ABB RAPID module: ST1606_R04_SWP_2.mod

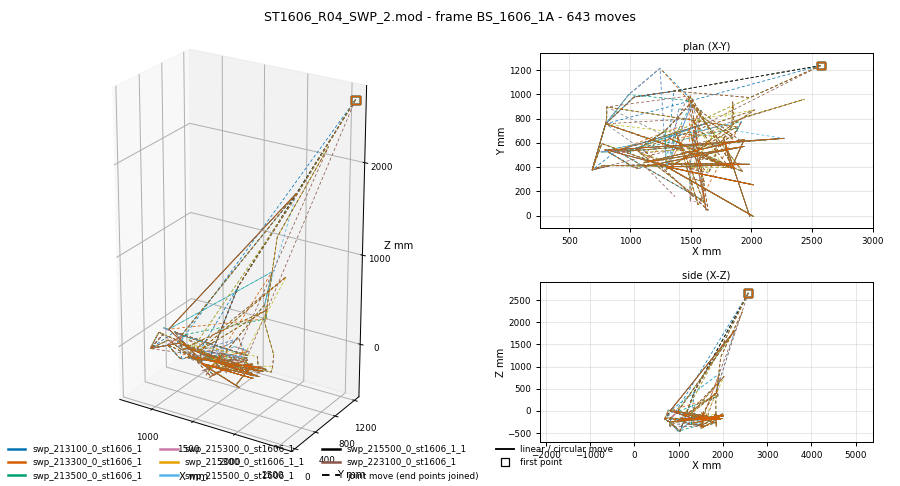
[picture p0: tool path of ST1606_R04_SWP_2.mod in frame BS_1606_1A, 643 of 1025 moves have a stored position in this frame; points joined in program order, loops and branches not executed]
MODULE ST1606_R04_SWP_2
CONST robtarget LHP_285:=[[1303.72,403.68,-203.75],[0.635635,0.00179403,0.00318194,-0.771981],[-1,-1,-1,0],[9E+09,9E+09,9E+09,9E+09,9E+09,9E+09]];
CONST robtarget LHP_275:=[[1301.19,402.05,-200.09],[0.6354,0.000830935,0.00305671,-0.772177],[-1,-1,-1,0],[9E+09,9E+09,9E+09,9E+09,9E+09,9E+09]];
CONST robtarget LHP_295:=[[1301.18,402.05,-200.09],[0.635399,0.000829977,0.00305677,-0.772177],[-1,-1,-1,0],[9E+09,9E+09,9E+09,9E+09,9E+09,9E+09]];
CONST robtarget LHP_270:=[[767.48,594.20,-155.47],[0.511232,-0.0380294,0.0384775,-0.857738],[-1,-1,-1,0],[9E+09,9E+09,9E+09,9E+09,9E+09,9E+09]];
CONST robtarget LHP_35:=[[946.51,280.68,-61.37],[0.681512,-0.0530703,0.0236717,-0.729496],[-1,-1,-1,0],[9E+09,9E+09,9E+09,9E+09,9E+09,9E+09]];
CONST robtarget LHP_76:=[[1001.84,541.68,-25.00],[0.296784,-0.0658707,0.043797,-0.951663],[-1,-1,0,0],[9E+09,9E+09,9E+09,9E+09,9E+09,9E+09]];
CONST robtarget LHP_80:=[[888.28,533.44,-4.12],[0.256081,-0.0828864,0.058088,-0.961342],[-1,-1,0,0],[9E+09,9E+09,9E+09,9E+09,9E+09,9E+09]];
CONST robtarget LHP_90:=[[990.54,532.98,-17.68],[0.294359,-0.0710943,0.0347938,-0.952411],[-1,-1,0,0],[9E+09,9E+09,9E+09,9E+09,9E+09,9E+09]];
CONST robtarget LHP_86:=[[888.43,535.56,-4.02],[0.256121,-0.0829008,0.0580729,-0.961331],[-1,-1,0,0],[9E+09,9E+09,9E+09,9E+09,9E+09,9E+09]];
CONST robtarget LHP_96:=[[1001.89,531.58,-24.98],[0.296786,-0.0658745,0.0437906,-0.951662],[-1,-1,0,0],[9E+09,9E+09,9E+09,9E+09,9E+09,9E+09]];
CONST robtarget LHP_120:=[[888.43,534.97,-4.06],[0.256117,-0.0828895,0.0580877,-0.961332],[-1,-1,0,0],[9E+09,9E+09,9E+09,9E+09,9E+09,9E+09]];
CONST robtarget LHP_130:=[[976.30,531.44,-18.23],[0.289518,-0.0722185,0.03693,-0.95373],[-1,-1,0,0],[9E+09,9E+09,9E+09,9E+09,9E+09,9E+09]];
CONST robtarget LHP_106:=[[818.07,526.79,7.37],[0.226549,-0.0825481,0.052721,-0.969062],[-1,-1,0,0],[9E+09,9E+09,9E+09,9E+09,9E+09,9E+09]];
CONST robtarget LHP_140:=[[813.23,540.09,5.50],[0.203616,-0.0600557,0.0553882,-0.975636],[-1,-1,0,0],[9E+09,9E+09,9E+09,9E+09,9E+09,9E+09]];
CONST robtarget LHP_305:=[[1315.92,428.20,-139.09],[0.644633,0.00162574,0.00306103,-0.764485],[-1,-1,-1,0],[9E+09,9E+09,9E+09,9E+09,9E+09,9E+09]];
CONST robtarget LHP_95:=[[1137.13,401.53,-148.24],[0.465302,0.0650512,0.0937079,-0.877771],[-1,-1,-1,0],[9E+09,9E+09,9E+09,9E+09,9E+09,9E+09]];
CONST robtarget LHP_30:=[[810.70,415.20,9.23],[0.639806,-0.0807189,0.0295354,-0.763715],[-1,-1,-1,0],[9E+09,9E+09,9E+09,9E+09,9E+09,9E+09]];
CONST robtarget LHP_75:=[[1074.27,512.60,-33.94],[0.333599,-0.0675086,0.0283306,-0.939868],[-1,-1,0,0],[9E+09,9E+09,9E+09,9E+09,9E+09,9E+09]];
CONST robtarget LHP_60:=[[1486.65,949.59,-335.01],[0.314,0.0992422,0.101035,-0.938801],[-1,-1,0,0],[9E+09,9E+09,9E+09,9E+09,9E+09,9E+09]];
CONST robtarget LHP_62:=[[1903.50,403.96,-168.40],[0.688588,0.0102129,0.00768242,-0.72504],[-1,-1,-1,0],[9E+09,9E+09,9E+09,9E+09,9E+09,9E+09]];
CONST robtarget LHP_061:=[[1899.73,616.36,-175.94],[0.688576,0.010205,0.00768425,-0.725052],[-1,-1,-1,0],[9E+09,9E+09,9E+09,9E+09,9E+09,9E+09]];
CONST robtarget LHP_602:=[[1726.06,605.49,-175.95],[0.68856,0.0102045,0.00768354,-0.725067],[-1,-1,-1,0],[9E+09,9E+09,9E+09,9E+09,9E+09,9E+09]];
CONST robtarget LHP_079:=[[2016.26,-5.68,-78.35],[0.747483,0.000532313,0.000430293,-0.664281],[-1,-1,-1,0],[9E+09,9E+09,9E+09,9E+09,9E+09,9E+09]];
CONST robtarget LHP_0792:=[[1914.27,375.53,-160.96],[0.711937,0.00638954,0.00588801,-0.702189],[-1,-1,-1,0],[9E+09,9E+09,9E+09,9E+09,9E+09,9E+09]];
CONST robtarget LHP_65:=[[1317.44,742.66,-303.72],[0.355107,0.0744104,0.10019,-0.926458],[-1,-1,0,0],[9E+09,9E+09,9E+09,9E+09,9E+09,9E+09]];
CONST robtarget LHP_85:=[[1629.29,310.10,-175.34],[0.669574,0.0105491,-0.00428905,-0.742658],[-1,0,-1,0],[9E+09,9E+09,9E+09,9E+09,9E+09,9E+09]];
CONST robtarget LHP_315:=[[1770.47,642.52,-185.25],[0.687362,-0.000165211,-0.0154473,-0.726151],[-1,0,-1,0],[9E+09,9E+09,9E+09,9E+09,9E+09,9E+09]];
CONST robtarget LHP_325:=[[1942.15,629.05,-193.52],[0.692101,-6.80423E-05,-0.0154578,-0.721635],[-1,0,-1,0],[9E+09,9E+09,9E+09,9E+09,9E+09,9E+09]];
CONST robtarget LHP_335:=[[1942.18,570.86,-193.52],[0.673118,-0.00046509,-0.0154488,-0.739373],[-1,0,-1,0],[9E+09,9E+09,9E+09,9E+09,9E+09,9E+09]];
CONST robtarget LHP_345:=[[1903.37,431.47,-166.61],[0.699368,0.00456834,-0.0108725,-0.714664],[-1,0,-1,0],[9E+09,9E+09,9E+09,9E+09,9E+09,9E+09]];
CONST robtarget LHP_355:=[[1863.39,397.38,-157.88],[0.649959,0.00383079,-0.0111584,-0.759877],[-1,0,-1,0],[9E+09,9E+09,9E+09,9E+09,9E+09,9E+09]];
CONST robtarget LHP_365:=[[1863.47,385.43,-144.48],[0.649789,-0.0155667,-0.0338777,-0.7592],[-1,0,-1,0],[9E+09,9E+09,9E+09,9E+09,9E+09,9E+09]];
CONST robtarget LHP_280:=[[2016.33,-5.64,-99.38],[0.747492,0.000549922,0.000436579,-0.664271],[-1,-1,-1,0],[9E+09,9E+09,9E+09,9E+09,9E+09,9E+09]];
CONST robtarget LHP_290:=[[2016.31,254.27,-112.69],[0.752523,0.000550496,0.000440421,-0.658565],[-1,-1,-1,0],[9E+09,9E+09,9E+09,9E+09,9E+09,9E+09]];
CONST robtarget LHP_300:=[[1984.86,424.01,-175.49],[0.757242,0.000550801,0.000441944,-0.653134],[-1,-1,-1,0],[9E+09,9E+09,9E+09,9E+09,9E+09,9E+09]];
CONST robtarget LHP_375:=[[1628.09,45.58,-117.32],[0.667896,0.00169065,-0.00043216,-0.744252],[-1,0,-1,0],[9E+09,9E+09,9E+09,9E+09,9E+09,9E+09]];
CONST robtarget LHP_385:=[[1611.54,278.38,-117.33],[0.667901,0.00169334,-0.000433516,-0.744248],[-1,0,-1,0],[9E+09,9E+09,9E+09,9E+09,9E+09,9E+09]];
CONST robtarget LHP_116:=[[1000.78,413.85,-25.10],[0.394135,-0.0875222,0.0272439,-0.91447],[-1,-1,0,0],[9E+09,9E+09,9E+09,9E+09,9E+09,9E+09]];
CONST robtarget LHP_150:=[[1561.93,87.92,-128.43],[0.625297,0.0429298,0.0210226,-0.778921],[-1,-1,-1,0],[9E+09,9E+09,9E+09,9E+09,9E+09,9E+09]];
CONST robtarget LHP_395:=[[1629.22,373.82,-175.87],[0.62292,0.0114274,-0.00461499,-0.782189],[-1,0,-1,0],[9E+09,9E+09,9E+09,9E+09,9E+09,9E+09]];
CONST robtarget LHP_405:=[[1666.92,623.72,-173.59],[0.685638,0.0117691,-0.00364924,-0.727838],[-1,0,-1,0],[9E+09,9E+09,9E+09,9E+09,9E+09,9E+09]];
CONST robtarget LHP_415:=[[1910.33,618.10,-173.56],[0.724769,0.0119478,-0.00298906,-0.688882],[-1,0,-1,0],[9E+09,9E+09,9E+09,9E+09,9E+09,9E+09]];
CONST robtarget LHP_425:=[[1929.29,361.85,-152.34],[0.724775,0.0119437,-0.00298739,-0.688875],[-1,0,-1,0],[9E+09,9E+09,9E+09,9E+09,9E+09,9E+09]];
CONST robtarget LHP_435:=[[1816.72,397.75,-147.92],[0.816486,0.00152322,-0.000785194,-0.577362],[-1,0,-1,0],[9E+09,9E+09,9E+09,9E+09,9E+09,9E+09]];
CONST robtarget LHP_310:=[[1987.44,-5.82,-69.73],[0.747483,0.000551369,0.000433351,-0.664281],[-1,-1,-1,0],[9E+09,9E+09,9E+09,9E+09,9E+09,9E+09]];
CONST robtarget LHP_445:=[[1643.36,44.45,-93.66],[0.669275,0.0117171,-0.00391081,-0.742912],[-1,0,-1,0],[9E+09,9E+09,9E+09,9E+09,9E+09,9E+09]];
CONST robtarget LHP_081:=[[1770.69,382.20,-42.12],[0.747485,0.000553614,0.00043516,-0.664279],[-1,-1,-1,0],[9E+09,9E+09,9E+09,9E+09,9E+09,9E+09]];
CONST robtarget LHP_320:=[[1834.77,390.06,-64.76],[0.679356,0.0474033,0.0375445,-0.731313],[-1,-1,-1,0],[9E+09,9E+09,9E+09,9E+09,9E+09,9E+09]];
CONST robtarget LHP_088:=[[1834.77,390.06,-64.76],[0.679356,0.0474033,0.0375445,-0.731313],[-1,-1,-1,0],[9E+09,9E+09,9E+09,9E+09,9E+09,9E+09]];
CONST robtarget LHP_97:=[[1624.62,82.13,-48.66],[0.622006,0.00520638,0.00406435,-0.782985],[-1,-1,-1,0],[9E+09,9E+09,9E+09,9E+09,9E+09,9E+09]];
LOCAL CONST robtarget LHP_089:=[[1624.62,82.13,-48.66],[0.622006,0.00520701,0.00406451,-0.782985],[-1,-1,-1,0],[9E+09,9E+09,9E+09,9E+09,9E+09,9E+09]];
CONST robtarget LHP_99:=[[1624.61,82.13,-48.66],[0.622006,0.00520638,0.00406435,-0.782985],[-1,-1,-1,0],[9E+09,9E+09,9E+09,9E+09,9E+09,9E+09]];
CONST robtarget LHP_109:=[[1624.62,82.13,-48.66],[0.622006,0.00520677,0.00406445,-0.782985],[-1,-1,-1,0],[9E+09,9E+09,9E+09,9E+09,9E+09,9E+09]];
CONST robtarget G0216022538BPS0:=[[2172.49,515.89,-41.57],[0.756815,0.0088806,0.00204198,-0.653566],[-1,-1,-1,0],[9E+09,9E+09,9E+09,9E+09,9E+09,9E+09]];
CONST robtarget LHP_40:=[[809.47,413.89,9.27],[0.637646,-0.0807527,0.029297,-0.765525],[-1,-1,-1,0],[9E+09,9E+09,9E+09,9E+09,9E+09,9E+09]];
CONST robtarget LHP_160:=[[1610.65,106.32,-46.18],[0.687963,0.00231302,0.000740632,-0.725741],[-1,-1,-1,0],[9E+09,9E+09,9E+09,9E+09,9E+09,9E+09]];
CONST robtarget LHP_126:=[[1076.78,394.51,-236.89],[0.363169,0.0511528,0.105229,-0.924347],[-1,-1,0,0],[9E+09,9E+09,9E+09,9E+09,9E+09,9E+09]];
CONST robtarget LHP_170:=[[2025.64,871.45,770.69],[0.675035,-0.0194872,0.00274828,-0.737523],[-1,0,-1,0],[9E+09,9E+09,9E+09,9E+09,9E+09,9E+09]];
CONST robtarget LHP_180:=[[1877.16,731.97,416.16],[0.599046,-0.0133068,0.00945685,-0.800548],[-1,-1,-1,0],[9E+09,9E+09,9E+09,9E+09,9E+09,9E+09]];
CONST robtarget LHP_190:=[[1874.96,717.56,328.63],[0.573795,-0.0241176,0.0161197,-0.818485],[-1,-1,-1,0],[9E+09,9E+09,9E+09,9E+09,9E+09,9E+09]];
CONST robtarget LHP_145:=[[1309.88,408.15,-170.82],[0.61629,0.069197,0.0627503,-0.78196],[-1,-1,-1,0],[9E+09,9E+09,9E+09,9E+09,9E+09,9E+09]];
CONST robtarget LHP_155:=[[1382.58,676.22,-177.76],[0.528172,0.00138203,0.0696209,-0.846277],[-1,-1,-1,0],[9E+09,9E+09,9E+09,9E+09,9E+09,9E+09]];
CONST robtarget LHP_165:=[[1054.33,541.75,-228.24],[0.365987,0.0660929,0.0753237,-0.925209],[-1,-1,0,0],[9E+09,9E+09,9E+09,9E+09,9E+09,9E+09]];
CONST robtarget LHP_175:=[[1299.24,382.14,-44.21],[0.616871,0.063591,0.0621051,-0.782029],[-1,-1,-1,0],[9E+09,9E+09,9E+09,9E+09,9E+09,9E+09]];
CONST robtarget LHP_50:=[[744.68,713.96,-233.05],[0.385967,0.0202354,0.0454893,-0.921168],[-1,-1,-1,0],[9E+09,9E+09,9E+09,9E+09,9E+09,9E+09]];
CONST robtarget LHP_136:=[[1076.49,400.39,-154.42],[0.36422,-0.00449082,0.0919532,-0.926751],[-1,-1,0,0],[9E+09,9E+09,9E+09,9E+09,9E+09,9E+09]];
CONST robtarget LHP_146:=[[1309.28,635.03,-261.94],[0.359345,0.128525,0.122572,-0.916149],[-1,-1,0,0],[9E+09,9E+09,9E+09,9E+09,9E+09,9E+09]];
CONST robtarget LHP_156:=[[1444.08,746.10,-205.80],[0.413851,0.0959699,0.0635629,-0.903038],[-1,-1,0,0],[9E+09,9E+09,9E+09,9E+09,9E+09,9E+09]];
CONST robtarget LHP_185:=[[1918.49,774.31,837.60],[0.611383,0.0296129,0.0513059,-0.789114],[-1,-1,-1,0],[9E+09,9E+09,9E+09,9E+09,9E+09,9E+09]];
CONST robtarget LHP_195:=[[1918.47,774.29,837.58],[0.611382,0.0296093,0.0513075,-0.789115],[-1,-1,-1,0],[9E+09,9E+09,9E+09,9E+09,9E+09,9E+09]];
CONST robtarget LHP_200:=[[1803.58,658.60,-169.59],[0.558228,0.00243716,0.011574,-0.829603],[-1,-1,-1,0],[9E+09,9E+09,9E+09,9E+09,9E+09,9E+09]];
CONST robtarget LHP_210:=[[1647.60,350.34,-198.93],[0.568544,0.0204485,0.0145518,-0.82227],[-1,-1,-1,0],[9E+09,9E+09,9E+09,9E+09,9E+09,9E+09]];
CONST robtarget LHP_70:=[[848.85,414.20,2.47],[0.587458,-0.0729773,0.0228571,-0.805634],[-1,-1,-1,0],[9E+09,9E+09,9E+09,9E+09,9E+09,9E+09]];
CONST robtarget LHP_205:=[[1074.21,512.85,-34.03],[0.333599,-0.0675174,0.0283721,-0.939866],[-1,-1,0,0],[9E+09,9E+09,9E+09,9E+09,9E+09,9E+09]];
CONST robtarget LHP_230:=[[1382.58,676.21,-177.77],[0.528172,0.00138131,0.0696207,-0.846277],[-1,-1,-1,0],[9E+09,9E+09,9E+09,9E+09,9E+09,9E+09]];
CONST robtarget LHP_215:=[[1878.70,697.76,491.72],[0.548791,-0.0233899,0.00387167,-0.835624],[-1,-1,-1,0],[9E+09,9E+09,9E+09,9E+09,9E+09,9E+09]];
CONST robtarget LHP_15:=[[1990.21,974.03,1486.76],[0.667208,-0.21865,0.214526,-0.678973],[-1,-1,-1,0],[9E+09,9E+09,9E+09,9E+09,9E+09,9E+09]];
CONST robtarget LHP_645:=[[1529.05,787.39,-322.41],[0.690547,-0.00133195,0.00252418,-0.723282],[-1,-1,-1,0],[9E+09,9E+09,9E+09,9E+09,9E+09,9E+09]];

PROC swp_213100_0_st1606_1()

! Lokale Hilfspunktdeklarationen
!=======================================
CONST robtarget LHP_000:=[[2573.53101,1238.19995,2660.84204],[0.56645757,-0.58473384,0.19941168,-0.54538715],[-1,-1,-1,4],[9E9,9E9,9E9,9E9,9E9,9E9]];
CONST robtarget LHP_005:=[[1360.172,1026.896,440.838989],[0.5866833,0.005191112,0.051883798,-0.80813605],[-1,-1,-1,0],[9E9,9E9,9E9,9E9,9E9,9E9]];
CONST robtarget LHP_010:=[[1032.36804,977.945984,-459.062988],[0.43703678,0.12694271,0.09414318,-0.8854499],[-1,-1,-1,0],[9E9,9E9,9E9,9E9,9E9,9E9]];
CONST robtarget LHP_015:=[[798.565002,757.20697,-251.078003],[0.47486252,-0.019805102,0.048932664,-0.87847537],[-1,-1,-1,0],[9E9,9E9,9E9,9E9,9E9,9E9]];
CONST robtarget LHP_020:=[[687.611023,377.389008,-182.513],[0.5033828,-0.04139257,0.03810638,-0.8622299],[-1,-1,-1,0],[9E9,9E9,9E9,9E9,9E9,9E9]];
CONST robtarget LHP_025:=[[830.614014,411.636993,5.70800018],[0.57761043,-0.07026652,0.026779216,-0.8128417],[-1,-1,-1,0],[9E9,9E9,9E9,9E9,9E9,9E9]];
CONST robtarget LHP_030:=[[774.456421,412.834808,12.8818998],[0.51775956,-0.07609037,0.018880999,-0.8519265],[-1,-1,-1,0],[9E9,9E9,9E9,9E9,9E9,9E9]];
CONST robtarget LHP_035:=[[687.669006,377.36499,-182.524002],[0.5034058,-0.04138605,0.0381097,-0.8622166],[-1,-1,-1,0],[9E9,9E9,9E9,9E9,9E9,9E9]];
CONST robtarget LHP_040:=[[798.562012,757.210999,-251.074997],[0.47486252,-0.019805102,0.048932664,-0.87847537],[-1,-1,-1,0],[9E9,9E9,9E9,9E9,9E9,9E9]];
CONST robtarget LHP_045:=[[989.937012,998.937012,-459.294006],[0.3557108,0.11797417,0.10516129,-0.9211368],[-1,-1,0,0],[9E9,9E9,9E9,9E9,9E9,9E9]];
CONST robtarget LHP_050:=[[1247.34399,1214.96399,-268.134003],[0.1820915,0.09153603,0.12369742,-0.97116566],[-1,-1,0,0],[9E9,9E9,9E9,9E9,9E9,9E9]];
CONST robtarget LHP_055:=[[1516.80,945.58,-312.06],[0.333537,0.109965,0.107679,-0.930089],[-1,-1,0,0],[9E+09,9E+09,9E+09,9E+09,9E+09,9E+09]];
CONST robtarget LHP_060:=[[1289.96,699.55,-313.54],[0.434357,0.0577433,0.142655,-0.887496],[-1,-1,0,0],[9E+09,9E+09,9E+09,9E+09,9E+09,9E+09]];
CONST robtarget LHP_065:=[[1054.38696,541.690002,-228.089005],[0.31436306,0.061803795,0.07883649,-0.9440026],[-1,-1,0,0],[9E9,9E9,9E9,9E9,9E9,9E9]];
CONST robtarget LHP_066:=[[1001.90,512.66,-24.97],[0.296786,-0.0658732,0.0437859,-0.951663],[-1,-1,0,0],[9E+09,9E+09,9E+09,9E+09,9E+09,9E+09]];
CONST robtarget LHP_070:=[[793.036987,542.02301,-179.692993],[0.20754133,0.019031575,0.0932444,-0.9735861],[-1,-1,0,0],[9E9,9E9,9E9,9E9,9E9,9E9]];
CONST robtarget LHP_075:=[[1029.48999,400.42099,-202.979004],[0.39562756,-0.007666591,0.14027788,-0.9076024],[-1,-1,0,0],[9E9,9E9,9E9,9E9,9E9,9E9]];
CONST robtarget LHP_076:=[[1000.77,413.90,-25.13],[0.39413,-0.0875132,0.0272435,-0.914473],[-1,-1,0,0],[9E+09,9E+09,9E+09,9E+09,9E+09,9E+09]];
CONST robtarget LHP_080:=[[1076.25195,387.731995,-208.341995],[0.43962634,0.059819497,0.10055306,-0.8905276],[-1,-1,0,0],[9E9,9E9,9E9,9E9,9E9,9E9]];
CONST robtarget LHP_085:=[[1115.20,414.51,-186.17],[0.4653,0.0650512,0.093708,-0.877772],[-1,-1,-1,0],[9E+09,9E+09,9E+09,9E+09,9E+09,9E+09]];
CONST robtarget LHP_090:=[[1309.86,408.19,-170.85],[0.635091,0.0676613,0.0644102,-0.766768],[-1,-1,-1,0],[9E+09,9E+09,9E+09,9E+09,9E+09,9E+09]];
CONST robtarget LHP_095:=[[1401.54,879.38,-183.06],[0.594946,-0.00205119,0.00205856,-0.80376],[-1,-1,-1,0],[9E+09,9E+09,9E+09,9E+09,9E+09,9E+09]];
CONST robtarget LHP_100:=[[1585.75903,868.737976,-184.042999],[0.62958896,-0.001844419,0.002234461,-0.776923],[-1,-1,-1,0],[9E9,9E9,9E9,9E9,9E9,9E9]];
CONST robtarget LHP_105:=[[1494.36597,427.148987,-193.410995],[0.49274465,0.06743884,0.029284334,-0.8670624],[-1,-1,-1,0],[9E9,9E9,9E9,9E9,9E9,9E9]];
CONST robtarget LHP_110:=[[1496.05298,118.202003,-107.422997],[0.51021767,0.050874773,0.015021431,-0.85840786],[-1,0,-1,0],[9E9,9E9,9E9,9E9,9E9,9E9]];
CONST robtarget LHP_115:=[[1617.51,116.05,-107.75],[0.656264,0.0400111,0.0250652,-0.753052],[-1,-1,-1,0],[9E+09,9E+09,9E+09,9E+09,9E+09,9E+09]];
CONST robtarget LHP_120:=[[1638.45496,381.700012,-207.240005],[0.5479616,0.037808824,0.05486916,-0.8338453],[-1,-1,-1,0],[9E9,9E9,9E9,9E9,9E9,9E9]];
CONST robtarget LHP_125:=[[1638.57495,764.435974,-176.789993],[0.56737936,0.11518183,0.1656212,-0.798363],[-1,-1,-1,0],[9E9,9E9,9E9,9E9,9E9,9E9]];
CONST robtarget LHP_130:=[[1832.91296,607.552002,669.677002],[0.6102957,-0.087358184,0.105843775,-0.78019536],[-1,-1,-1,0],[9E9,9E9,9E9,9E9,9E9,9E9]];
CONST robtarget LHP_135:=[[2270.29395,637.606995,1817.37305],[0.6669749,-0.3265057,0.039168768,-0.6685838],[-1,-1,-1,0],[9E9,9E9,9E9,9E9,9E9,9E9]];

!****************************************************
!* Unterprogramm  : swp_213100_0_st1606_1           *
!* Modell/Typ     : FHS T3,5 R1 (3250mm)            *
!* Applikation    : Punktschweissen Zange 1         *
!* Anlagen/Station: Linie 16 / St1606               *
!* Robotername    : 1606R04                         *
!* Originalautor  : COMAU                           *
!* Erstelldatum   : 28.02.2006                      *
!****************************************************
!*               Aktualisierungen                   *
!*             ====================                 *
!* Datum       : 13.01.2017                         *
!* dz?nderung    : VS30 - Winter PU 2016/17           *
!* Gedz?ndert von: R. Ddz?rrbeck (ese-robotics fdz?r FFT) *
!****************************************************

 INIT_SW_BASE;

 WKZ_1_AUFNEHMEN;

 MoveJ ToolHome1,vSchnell,fine,nomtcp1;

 KOLLISION_ZONE 10\Anfrage;
 KOLLISION_ZONE 11\Anfrage;

 MoveJ LHP_000,vSchnell,fine,nomtcp1\WObj:=BS_1606_1A;
 Vorhub\auf;

 ! Warte auf Freigabe SPS, Fahrzeug in Position
 ABL 2\ABL_WAIT;
 ABL 10\ABL_SET;

!
! ZMIANA !!!
!
! Zmiana kolejnosci grzania
! Zrobic dojazd
WaitUntil FALSE;

 KOLLISION_ZONE 1\Anfrage;
 KOLLISION_ZONE 2\Anfrage;
 KOLLISION_ZONE 5\Anfrage;
 KOLLISION_ZONE 6\Anfrage;

 MoveJ LHP_040,vSchnell,z100,nomtcp1\WObj:=BS_1606_1A;
 MoveJ LHP_045,vSchnell,z100,nomtcp1\WObj:=BS_1606_1A;
 MoveJ LHP_050,vSchnell,z100,nomtcp1\WObj:=BS_1606_1A;
 MoveJ LHP_055,vSchnell,z100,nomtcp1\WObj:=BS_1606_1A;
 MoveJ LHP_060,vSchnell,z100,nomtcp1\WObj:=BS_1606_1A;
 MoveJ LHP_065,vSchnell,z100,nomtcp1\WObj:=BS_1606_1A;

 SpotL G0216020160BP20\VFO:=210,vSpot,nomtcp1\WObj:=BS_1606_1A;

 KOLLISION_ZONE 1\Freigabe;

 SpotL G0216020158BP20\VFO:=210,vSpot,nomtcp1\WObj:=BS_1606_1A;

 MoveL LHP_066,vSpot,z1,nomtcp1\WObj:=BS_1606_1A;
 MoveL [[1001.84,541.68,-25.00],[0.296784,-0.0658709,0.0437966,-0.951663],[-1,-1,0,0],[9E+09,9E+09,9E+09,9E+09,9E+09,9E+09]], vSpot, z1, nomtcp1\WObj:=BS_1606_1A;
 MoveL [[888.48,538.76,-4.07],[0.256126,-0.0828936,0.0580825,-0.961329],[-1,-1,0,0],[9E+09,9E+09,9E+09,9E+09,9E+09,9E+09]], vSpot, z1, nomtcp1\WObj:=BS_1606_1A;

 SpotL G0216020154BP20\VFO:=210,vSpot,nomtcp1\WObj:=BS_1606_1A;

 SpotL G0216020152BP20\VFO:=210,vSpot,nomtcp1\WObj:=BS_1606_1A;

 SpotL G0216020150BP20\VFO:=210,vSpot,nomtcp1\WObj:=BS_1606_1A;
 MoveL [[823.31,527.82,7.40],[0.226542,-0.0825543,0.0527166,-0.969064],[-1,-1,0,0],[9E+09,9E+09,9E+09,9E+09,9E+09,9E+09]], vSpot, z1, nomtcp1\WObj:=BS_1606_1A;
 MoveL [[762.43,528.71,12.54],[0.205864,-0.0816335,0.0516713,-0.9738],[-1,-1,0,0],[9E+09,9E+09,9E+09,9E+09,9E+09,9E+09]], vSpot, z1, nomtcp1\WObj:=BS_1606_1A;

 SpotL G0216047004BP20\VFO:=210\Vorhub_Auf,vSpot,nomtcp1\WObj:=BS_1606_1A;

 MoveJ LHP_070,vSchnell,z100,nomtcp1\WObj:=BS_1606_1A;
 MoveJ LHP_075,vSchnell,z100,nomtcp1\WObj:=BS_1606_1A;

 SpotL G0216020168BP20\VFO:=210,vSpot,nomtcp1\WObj:=BS_1606_1A;

 MoveL LHP_076,vSpot,z1,nomtcp1\WObj:=BS_1606_1A;

 SpotL G0216020164BP20\VFO:=210,vSpot,nomtcp1\WObj:=BS_1606_1A;

!SWP neue Koordinaden
 MoveL LHP_076,vSpot,z1,nomtcp1\WObj:=BS_1606_1A;

 SpotL G0216020162BP20\VFO:=210\Vorhub_Auf,vSpot,nomtcp1\WObj:=BS_1606_1A;
 MoveJ LHP_116, vSpot, z1, nomtcp1\WObj:=BS_1606_1A;

 MoveJ LHP_080,vSchnell,z100,nomtcp1\WObj:=BS_1606_1A;
 MoveJ LHP_085,vSchnell,z100,nomtcp1\WObj:=BS_1606_1A;
 MoveL [[1300.37,401.52,-167.52],[0.611248,0.080394,0.0809277,-0.783175],[-1,-1,-1,0],[9E+09,9E+09,9E+09,9E+09,9E+09,9E+09]], vSchnell, z10, nomtcp1\WObj:=BS_1606_1A;
 MoveL [[1299.24,382.15,-44.23],[0.616868,0.0635976,0.0621051,-0.78203],[-1,-1,-1,0],[9E+09,9E+09,9E+09,9E+09,9E+09,9E+09]], vSchnell, z10, nomtcp1\WObj:=BS_1606_1A;

 !
 ! ZMIANA !!!
 !
 ! Te punkty byly robione jako pierwsze
 !
 WaitUntil FALSE;
 KOLLISION_ZONE 12 \Anfrage;

 MoveJ LHP_005,vSchnell,z100,nomtcp1\WObj:=BS_1606_1A;
 MoveJ LHP_010,vSchnell,z100,nomtcp1\WObj:=BS_1606_1A;
 MoveJ LHP_015,vSchnell,z100,nomtcp1\WObj:=BS_1606_1A;
 MoveJ LHP_020,vSchnell,z100,nomtcp1\WObj:=BS_1606_1A;

 SpotL G0216047007BP20\VFO:=210,vSpot,nomtcp1\WObj:=BS_1606_1A;
 MoveL LHP_025,vSchnell,z100,nomtcp1\WObj:=BS_1606_1A;

!SWP neue Koordinaden

 SpotL G0216020172BP20\VFO:=210,vSpot,nomtcp1\WObj:=BS_1606_1A;

 SpotL G0216020170BP20\VFO:=210\Vorhub_Auf,vSpot,nomtcp1\WObj:=BS_1606_1A;

 MoveL LHP_025,vSchnell,z100,nomtcp1\WObj:=BS_1606_1A;
 MoveJ LHP_030,vSchnell,z100,nomtcp1\WObj:=BS_1606_1A;
 MoveJ LHP_035,vSchnell,z100,nomtcp1\WObj:=BS_1606_1A;

 !
 ! ZMIANA!!!!!
 ! Powrot do HOME
 !

 WaitUntil FALSE;
 !SpotL G0216020180BP20\VFO:=210\Vorhub_Auf,vSpot,nomtcp1\WObj:=BS_1606_1A;

! MoveL [[1299.24,382.15,-44.23],[0.616868,0.0635976,0.0621051,-0.78203],[-1,-1,-1,0],[9E+09,9E+09,9E+09,9E+09,9E+09,9E+09]], vSchnell, z10, nomtcp1\WObj:=BS_1606_1A;
! MoveL [[1300.37,401.52,-167.52],[0.611248,0.080394,0.0809277,-0.783175],[-1,-1,-1,0],[9E+09,9E+09,9E+09,9E+09,9E+09,9E+09]], vSchnell, z10, nomtcp1\WObj:=BS_1606_1A;
! MoveJ LHP_090,vSchnell,z100,nomtcp1\WObj:=BS_1606_1A;
! MoveJ LHP_095,vSchnell,z100,nomtcp1\WObj:=BS_1606_1A;
! MoveJ LHP_100,vSchnell,z100,nomtcp1\WObj:=BS_1606_1A;
! MoveJ LHP_105,vSchnell,z100,nomtcp1\WObj:=BS_1606_1A;

! SpotL G0216020344BP20\VFO:=210,vSpot,nomtcp1\WObj:=BS_1606_1A;

! SpotL G0216020348BP20\VFO:=210,vSpot,nomtcp1\WObj:=BS_1606_1A;
! SpotL G0216020352BP20\VFO:=210\Vorhub_Auf,vSpot,nomtcp1\WObj:=BS_1606_1A;

! MoveJ LHP_110,vSchnell,z100,nomtcp1\WObj:=BS_1606_1A;
! MoveJ LHP_150, vSchnell, z100, nomtcp1\WObj:=BS_1606_1A;


 !Start Kollision mit Skid ! (Folie81)
! MoveJ LHP_115,vSchnell,z100,nomtcp1\WObj:=BS_1606_1A;
 !Ende Kollision mit Skid ! (Folie81)

 !Start Kollision mit Skid ! (Folie82)
! SpotL G0216020358BP20\VFO:=210,vSpot,nomtcp1\WObj:=BS_1606_1A;
 !Ende Kollision mit Skid ! (Folie82)
! SpotL G0216020366BP20\VFO:=210\Vorhub_Auf,vSpot,nomtcp1\WObj:=BS_1606_1A;

 MoveJ LHP_120,vSchnell,z100,nomtcp1\WObj:=BS_1606_1A;
 MoveJ LHP_125,vSchnell,z100,nomtcp1\WObj:=BS_1606_1A;
 MoveJ LHP_130,vSchnell,z100,nomtcp1\WObj:=BS_1606_1A;
 MoveJ LHP_135,vSchnell,z100,nomtcp1\WObj:=BS_1606_1A;

 MoveJ ToolHome1,vSchnell,fine,nomtcp1;

 KOLLISION_ZONE 2\Freigabe;
 KOLLISION_ZONE 5\Freigabe;
 KOLLISION_ZONE 6\Freigabe;
 KOLLISION_ZONE 10\Freigabe;
 KOLLISION_ZONE 11\Freigabe;
 KOLLISION_ZONE 12\Freigabe;

 ! Warte auf Freigabe SPS, Fertigmeldung Schweissen
 ABL 254\ABL_WAIT;
 ABL 255\ABL_SET;

ENDPROC !Punktschweissen Zange 1, FHS T3,5 R1 (3250mm)


PROC swp_213300_0_st1606_1()

! Lokale Hilfspunktdeklarationen
!=======================================
CONST robtarget LHP_000:=[[2573.528,1238.2,2660.84],[0.56645757,-0.58473384,0.19941168,-0.54538715],[-1,-1,-1,4],[9E9,9E9,9E9,9E9,9E9,9E9]];
CONST robtarget LHP_005:=[[1247.39,1136.00,760.30],[0.5238,-0.0971482,0.0777334,-0.842706],[-1,-1,-1,0],[9E+09,9E+09,9E+09,9E+09,9E+09,9E+09]];
CONST robtarget LHP_010:=[[1032.368,977.946,-459.063],[0.43703678,0.12694271,0.09414318,-0.8854499],[-1,-1,-1,0],[9E9,9E9,9E9,9E9,9E9,9E9]];
CONST robtarget LHP_015:=[[798.565,757.207,-251.078],[0.47486252,-0.019805102,0.048932664,-0.87847537],[-1,-1,-1,0],[9E9,9E9,9E9,9E9,9E9,9E9]];
CONST robtarget LHP_020:=[[687.611,377.389,-182.513],[0.5033828,-0.04139257,0.03810638,-0.8622299],[-1,-1,-1,0],[9E9,9E9,9E9,9E9,9E9,9E9]];
CONST robtarget LHP_025:=[[830.614,411.637,5.708],[0.57761043,-0.07026652,0.026779216,-0.8128417],[-1,-1,-1,0],[9E9,9E9,9E9,9E9,9E9,9E9]];
CONST robtarget LHP_030:=[[774.461,412.833,16.893],[0.51776165,-0.076091945,0.018879995,-0.85192513],[-1,-1,-1,0],[9E9,9E9,9E9,9E9,9E9,9E9]];
CONST robtarget LHP_035:=[[687.669,377.365,-182.524],[0.5034058,-0.04138605,0.0381097,-0.8622166],[-1,-1,-1,0],[9E9,9E9,9E9,9E9,9E9,9E9]];
CONST robtarget LHP_040:=[[798.562,757.211,-251.075],[0.47486252,-0.019805102,0.048932664,-0.87847537],[-1,-1,-1,0],[9E9,9E9,9E9,9E9,9E9,9E9]];
CONST robtarget LHP_045:=[[989.937,998.937,-459.294],[0.3557108,0.11797417,0.10516129,-0.9211368],[-1,-1,0,0],[9E9,9E9,9E9,9E9,9E9,9E9]];
CONST robtarget LHP_050:=[[1247.344,1214.964,-268.134],[0.1820915,0.09153603,0.12369742,-0.97116566],[-1,-1,0,0],[9E9,9E9,9E9,9E9,9E9,9E9]];
CONST robtarget LHP_055:=[[1280.56,716.07,-303.30],[0.431068,0.0952157,0.0788807,-0.893808],[-1,-1,0,0],[9E+09,9E+09,9E+09,9E+09,9E+09,9E+09]];
CONST robtarget LHP_060:=[[1126.92,615.76,-282.67],[0.360168,0.0736591,0.0772281,-0.926763],[-1,-1,0,0],[9E+09,9E+09,9E+09,9E+09,9E+09,9E+09]];
CONST robtarget LHP_065:=[[1058.91,591.54,-248.55],[0.324693,0.0626502,0.0781167,-0.940504],[-1,-1,0,0],[9E+09,9E+09,9E+09,9E+09,9E+09,9E+09]];
CONST robtarget LHP_066:=[[1001.90,512.66,-24.97],[0.296786,-0.0658732,0.0437859,-0.951663],[-1,-1,0,0],[9E+09,9E+09,9E+09,9E+09,9E+09,9E+09]];
CONST robtarget LHP_070:=[[990.55,511.98,-17.63],[0.29436,-0.0711019,0.0347764,-0.952411],[-1,-1,0,0],[9E+09,9E+09,9E+09,9E+09,9E+09,9E+09]];
CONST robtarget LHP_075:=[[793.037,542.023,-179.693],[0.20754133,0.019031575,0.0932444,-0.9735861],[-1,-1,0,0],[9E9,9E9,9E9,9E9,9E9,9E9]];
CONST robtarget LHP_080:=[[1029.49,400.421,-202.979],[0.39562756,-0.007666591,0.14027788,-0.9076024],[-1,-1,0,0],[9E9,9E9,9E9,9E9,9E9,9E9]];
CONST robtarget LHP_085:=[[913.891,403.285,-23.344],[0.33140895,-0.07444555,0.018514868,-0.94036335],[-1,-1,0,0],[9E9,9E9,9E9,9E9,9E9,9E9]];
CONST robtarget LHP_086:=[[1000.76,413.91,-25.16],[0.378586,-0.0879607,0.0257669,-0.921017],[-1,-1,0,0],[9E+09,9E+09,9E+09,9E+09,9E+09,9E+09]];
CONST robtarget LHP_090:=[[1076.252,387.732,-208.342],[0.43962634,0.059819497,0.10055306,-0.8905276],[-1,-1,0,0],[9E9,9E9,9E9,9E9,9E9,9E9]];
CONST robtarget LHP_095:=[[1115.20,414.51,-186.17],[0.4653,0.0650512,0.093708,-0.877772],[-1,-1,-1,0],[9E+09,9E+09,9E+09,9E+09,9E+09,9E+09]];
CONST robtarget LHP_100:=[[1309.89,408.15,-170.80],[0.616296,0.0691966,0.0627474,-0.781955],[-1,-1,-1,0],[9E+09,9E+09,9E+09,9E+09,9E+09,9E+09]];
CONST robtarget LHP_105:=[[1403.48,885.26,-182.95],[0.551408,-0.0122764,0.0175739,-0.83396],[-1,-1,-1,0],[9E+09,9E+09,9E+09,9E+09,9E+09,9E+09]];
CONST robtarget LHP_110:=[[1382.58,676.23,-177.75],[0.52817,0.00138314,0.0696209,-0.846279],[-1,-1,-1,0],[9E+09,9E+09,9E+09,9E+09,9E+09,9E+09]];
CONST robtarget LHP_115:=[[1516.89,728.30,-174.24],[0.498509,0.0194939,0.0152407,-0.866532],[-1,-1,-1,0],[9E+09,9E+09,9E+09,9E+09,9E+09,9E+09]];
CONST robtarget LHP_120:=[[1494.68,367.84,-180.88],[0.523408,0.0111235,0.00571408,-0.851991],[-1,-1,-1,0],[9E+09,9E+09,9E+09,9E+09,9E+09,9E+09]];
CONST robtarget LHP_125:=[[1516.99,109.79,-122.77],[0.510502,0.031993,0.0287635,-0.8588],[-1,-1,-1,0],[9E+09,9E+09,9E+09,9E+09,9E+09,9E+09]];
CONST robtarget LHP_130:=[[1619.68,161.21,-115.86],[0.5571,0.0367268,0.0384586,-0.828741],[-1,-1,-1,0],[9E+09,9E+09,9E+09,9E+09,9E+09,9E+09]];
CONST robtarget LHP_135:=[[1647.59,350.35,-198.92],[0.568544,0.0204469,0.0145536,-0.82227],[-1,-1,-1,0],[9E+09,9E+09,9E+09,9E+09,9E+09,9E+09]];
CONST robtarget LHP_140:=[[1803.57,658.62,-169.58],[0.558227,0.00243614,0.0115763,-0.829604],[-1,-1,-1,0],[9E+09,9E+09,9E+09,9E+09,9E+09,9E+09]];
CONST robtarget LHP_145:=[[2025.676,871.423,770.799],[0.69849163,-0.019397179,0.003350246,-0.7153474],[-1,0,-1,0],[9E9,9E9,9E9,9E9,9E9,9E9]];
CONST robtarget LHP_150:=[[2270.286,637.595,1817.362],[0.66697776,-0.32649988,0.039162926,-0.6685841],[-1,-1,-1,0],[9E9,9E9,9E9,9E9,9E9,9E9]];

!****************************************************
!* Unterprogramm  : swp_213300_0_st1606_1           *
!* Modell/Typ     : FHS T3,5 R2 (3665mm)            *
!* Applikation    : Punktschweissen Zange 1         *
!* Anlagen/Station: Linie 16 / St1606               *
!* Robotername    : 1606R04                         *
!* Originalautor  : COMAU                           *
!* Erstelldatum   : 28.02.2006                      *
!****************************************************
!*               Aktualisierungen                   *
!*             ====================                 *
!* Datum       : 13.01.2017                         *
!* dz?nderung    : VS30 - Winter PU 2016/17           *
!* Gedz?ndert von: R. Ddz?rrbeck (ese-robotics fdz?r FFT) *
!****************************************************

 INIT_SW_BASE;

 WKZ_1_AUFNEHMEN;

 MoveJ ToolHome1,vSchnell,fine,nomtcp1;


 MoveJ LHP_000,vSchnell,fine,nomtcp1\WObj:=BS_1606_1A;
 Vorhub\auf;

 ! Warte auf Freigabe SPS, Fahrzeug in Position
 ABL 2\ABL_WAIT;
 ABL 10\ABL_SET;


 KOLLISION_ZONE 1\Anfrage;
 KOLLISION_ZONE 2\Anfrage;
 KOLLISION_ZONE 5\Anfrage;
 KOLLISION_ZONE 6\Anfrage;

 MoveJ LHP_005,vSchnell,z100,nomtcp1\WObj:=BS_1606_1A;
 MoveJ LHP_010,vSchnell,z100,nomtcp1\WObj:=BS_1606_1A;
 MoveJ LHP_015,vSchnell,z100,nomtcp1\WObj:=BS_1606_1A;
 MoveJ LHP_020,vSchnell,z100,nomtcp1\WObj:=BS_1606_1A;

 SpotL G0216047007BP20\VFO:=210, vSpot, nomtcp1\WObj:=BS_1606_1A;

!SWP neue Koordinaden

 SpotL G0216020172BP20\VFO:=210, vSpot, nomtcp1\WObj:=BS_1606_1A;

 SpotL G0216020170BP20\VFO:=210\Vorhub_Auf, vSpot, nomtcp1\WObj:=BS_1606_1A;

 MoveL LHP_025,vSchnell,z100,nomtcp1\WObj:=BS_1606_1A;
 MoveJ LHP_030,vSchnell,z100,nomtcp1\WObj:=BS_1606_1A;
 MoveJ LHP_035,vSchnell,z100,nomtcp1\WObj:=BS_1606_1A;
 MoveJ LHP_040,vSchnell,z100,nomtcp1\WObj:=BS_1606_1A;
 MoveJ LHP_045, vSchnell, fine, nomtcp1\WObj:=BS_1606_1A;
 KOLLISION_ZONE 1\Freigabe;
 MoveJ LHP_050,vSchnell,z100,nomtcp1\WObj:=BS_1606_1A;
 MoveJ LHP_60, vSchnell, z100, nomtcp1\WObj:=BS_1606_1A;
 !
 MoveJ LHP_110, vSchnell, fine, nomtcp1\WObj:=BS_1606_1A;
 MoveJ LHP_100,vSchnell,z100,nomtcp1\WObj:=BS_1606_1A;
 MoveL [[1300.37,401.52,-167.52],[0.611248,0.080394,0.0809277,-0.783175],[-1,-1,-1,0],[9E+09,9E+09,9E+09,9E+09,9E+09,9E+09]], vSchnell, z10, nomtcp1\WObj:=BS_1606_1A;
 MoveL [[1299.24,382.15,-44.23],[0.616868,0.0635976,0.0621051,-0.78203],[-1,-1,-1,0],[9E+09,9E+09,9E+09,9E+09,9E+09,9E+09]], vSchnell, z15, nomtcp1\WObj:=BS_1606_1A;
 !versch
 !
 ! ZMIANA !!!!
 !
 WaitUntil FALSE;
 !SpotL G0216020180BP20\VFO:=210\Vorhub_Auf, vSpot, nomtcp1\WObj:=BS_1606_1A;
 !
 MoveL [[1299.24,382.15,-44.23],[0.616868,0.0635976,0.0621051,-0.78203],[-1,-1,-1,0],[9E+09,9E+09,9E+09,9E+09,9E+09,9E+09]], vSchnell, z10, nomtcp1\WObj:=BS_1606_1A;
 MoveJ [[1300.37,401.52,-167.52],[0.611248,0.080394,0.0809277,-0.783175],[-1,-1,-1,0],[9E+09,9E+09,9E+09,9E+09,9E+09,9E+09]], vSchnell, z10, nomtcp1\WObj:=BS_1606_1A;
 !
 MoveJ [[1054.36,541.70,-228.11],[0.366013,0.0660625,0.0753086,-0.925202],[-1,-1,0,0],[9E+09,9E+09,9E+09,9E+09,9E+09,9E+09]], vSchnell, z10, nomtcp1\WObj:=BS_1606_1A;

 SpotL G0216020160BP20\VFO:=210, vSpot, nomtcp1\WObj:=BS_1606_1A;

 !KOLLISION_ZONE 1\Freigabe;


 SpotL G0216020158BP20\VFO:=210, vSpot, nomtcp1\WObj:=BS_1606_1A;
 !z2 frei moglich

 MoveL LHP_066,vSpot,z1,nomtcp1\WObj:=BS_1606_1A;
 MoveJ LHP_070,vSchnell,z100,nomtcp1\WObj:=BS_1606_1A;
 MoveL [[990.54,532.98,-17.68],[0.29436,-0.0710946,0.0347935,-0.952411],[-1,-1,0,0],[9E+09,9E+09,9E+09,9E+09,9E+09,9E+09]], vSchnell, z100, nomtcp1\WObj:=BS_1606_1A;
 MoveL [[888.28,533.44,-4.12],[0.256081,-0.0828865,0.0580874,-0.961342],[-1,-1,0,0],[9E+09,9E+09,9E+09,9E+09,9E+09,9E+09]], vSchnell, z100, nomtcp1\WObj:=BS_1606_1A;

 SpotL G0216020154BP20\VFO:=210, vSpot, nomtcp1\WObj:=BS_1606_1A;
 !
 KOLLISION_ZONE 2\Freigabe;

 SpotL G0216020152BP20\VFO:=210, vSpot, nomtcp1\WObj:=BS_1606_1A;

 SpotL G0216020150BP20\VFO:=210, vSpot, nomtcp1\WObj:=BS_1606_1A;
 MoveL [[818.05,527.90,7.41],[0.226537,-0.0825529,0.0527157,-0.969065],[-1,-1,0,0],[9E+09,9E+09,9E+09,9E+09,9E+09,9E+09]], vSchnell, z100, nomtcp1\WObj:=BS_1606_1A;
 MoveL [[762.43,526.03,12.55],[0.205854,-0.0816331,0.0516654,-0.973802],[-1,-1,0,0],[9E+09,9E+09,9E+09,9E+09,9E+09,9E+09]], vSchnell, z100, nomtcp1\WObj:=BS_1606_1A;

 SpotL G0216047004BP20\VFO:=210\Vorhub_Auf, vSpot, nomtcp1\WObj:=BS_1606_1A;

 MoveJ LHP_075,vSchnell,z100,nomtcp1\WObj:=BS_1606_1A;
 MoveJ LHP_080,vSchnell,z100,nomtcp1\WObj:=BS_1606_1A;
 MoveJ LHP_085,vSchnell,z100,nomtcp1\WObj:=BS_1606_1A;

 SpotL G0216020168BP20\VFO:=210, vSpot, nomtcp1\WObj:=BS_1606_1A;
 !z2 frei

 MoveL LHP_086,vSpot,z1,nomtcp1\WObj:=BS_1606_1A;

 SpotL G0216020164BP20\VFO:=210, vSpot, nomtcp1\WObj:=BS_1606_1A;

!SWP neue Koordinaden

 SpotL G0216020162BP20\VFO:=210\Vorhub_Auf, vSpot, nomtcp1\WObj:=BS_1606_1A;

 !Start Kollision mit Skid ! (Folie74)
 MoveJ [[1076.49,400.40,-154.41],[0.36422,-0.00449148,0.0919521,-0.926752],[-1,-1,0,0],[9E+09,9E+09,9E+09,9E+09,9E+09,9E+09]], vSpot, z100, nomtcp1\WObj:=BS_1606_1A;
 MoveJ [[1313.90,629.03,-259.50],[0.3607,0.127838,0.12237,-0.915739],[-1,-1,0,0],[9E+09,9E+09,9E+09,9E+09,9E+09,9E+09]], vSpot, z100, nomtcp1\WObj:=BS_1606_1A;
 MoveJ [[1444.08,746.07,-205.75],[0.41386,0.095959,0.0635554,-0.903035],[-1,-1,0,0],[9E+09,9E+09,9E+09,9E+09,9E+09,9E+09]], vSchnell, z100, nomtcp1\WObj:=BS_1606_1A;
 !


 !
 MoveJ LHP_120,vSchnell,z100,nomtcp1\WObj:=BS_1606_1A;

 SpotL G0216020668BP20\VFO:=210,vSpot,nomtcp1\WObj:=BS_1606_1A;


 SpotL G0216020670BP20\VFO:=210,vSpot,nomtcp1\WObj:=BS_1606_1A;
 SpotL G0216020674BP20\VFO:=210,vSpot,nomtcp1\WObj:=BS_1606_1A;
 SpotL G0216020676BP20\VFO:=210\Vorhub_Auf,vSpot,nomtcp1\WObj:=BS_1606_1A;

 MoveJ LHP_125,vSchnell,z100,nomtcp1\WObj:=BS_1606_1A;


 MoveJ LHP_130,vSchnell,z100,nomtcp1\WObj:=BS_1606_1A;

 SpotL G0216020682BP20\VFO:=210,vSpot,nomtcp1\WObj:=BS_1606_1A;

 SpotL G0216020684BP20\VFO:=210,vSpot,nomtcp1\WObj:=BS_1606_1A;
 SpotL G0216020686BP20\VFO:=210,vSpot,nomtcp1\WObj:=BS_1606_1A;
 SpotL G0216020688BP20\VFO:=210\Vorhub_Auf,vSpot,nomtcp1\WObj:=BS_1606_1A;

 MoveJ LHP_135,vSchnell,z100,nomtcp1\WObj:=BS_1606_1A;
 MoveJ LHP_140, vSchnell, fine, nomtcp1\WObj:=BS_1606_1A;
 KOLLISION_ZONE 5\Freigabe;
 !Z2\Frei;
 MoveJ [[1890.63,724.74,327.70],[0.573801,-0.0241184,0.0161214,-0.818481],[-1,-1,-1,0],[9E+09,9E+09,9E+09,9E+09,9E+09,9E+09]], vSchnell, z100, nomtcp1\WObj:=BS_1606_1A;
 MoveJ [[1878.66,697.77,491.79],[0.548782,-0.0234003,0.00386231,-0.835629],[-1,-1,-1,0],[9E+09,9E+09,9E+09,9E+09,9E+09,9E+09]], vSchnell, z100, nomtcp1\WObj:=BS_1606_1A;
 MoveJ [[1918.50,774.31,837.60],[0.611384,0.0296159,0.0513029,-0.789114],[-1,-1,-1,0],[9E+09,9E+09,9E+09,9E+09,9E+09,9E+09]], vSchnell, z100, nomtcp1\WObj:=BS_1606_1A;
 !MoveJ LHP_145,vSchnell,z100,nomtcp1\WObj:=BS_1606_1A;
 MoveJ LHP_150,vSchnell,z100,nomtcp1\WObj:=BS_1606_1A;

 MoveJ ToolHome1,vSchnell,fine,nomtcp1;

 !Z5\Frei;
 KOLLISION_ZONE 6\Freigabe;

 ! Warte auf Freigabe SPS, Fertigmeldung Schweissen
 ABL 254\ABL_WAIT;
 ABL 255\ABL_SET;
 !
 !

ENDPROC
 !Punktschweissen Zange 1, FHS T3,5 R2 (3665mm)

PROC swp_213500_0_st1606_1()

! Lokale Hilfspunktdeklarationen
!=======================================
CONST robtarget LHP_000:=[[2573.528,1238.2,2660.841],[0.56645757,-0.58473384,0.19941168,-0.54538715],[-1,-1,-1,4],[9E9,9E9,9E9,9E9,9E9,9E9]];
CONST robtarget LHP_005:=[[1360.172,1026.896,440.839],[0.5866833,0.005191112,0.051883798,-0.80813605],[-1,-1,-1,0],[9E9,9E9,9E9,9E9,9E9,9E9]];
CONST robtarget LHP_010:=[[1032.368,977.946,-459.063],[0.43703678,0.12694271,0.09414318,-0.8854499],[-1,-1,-1,0],[9E9,9E9,9E9,9E9,9E9,9E9]];
CONST robtarget LHP_015:=[[798.565,757.207,-251.078],[0.47486252,-0.019805102,0.048932664,-0.87847537],[-1,-1,-1,0],[9E9,9E9,9E9,9E9,9E9,9E9]];
CONST robtarget LHP_020:=[[687.611,377.389,-182.513],[0.5033828,-0.04139257,0.03810638,-0.8622299],[-1,-1,-1,0],[9E9,9E9,9E9,9E9,9E9,9E9]];
CONST robtarget LHP_025:=[[830.614,411.637,5.708],[0.57761043,-0.07026652,0.026779216,-0.8128417],[-1,-1,-1,0],[9E9,9E9,9E9,9E9,9E9,9E9]];
CONST robtarget LHP_030:=[[774.52,412.85,8.85],[0.517766,-0.0760768,0.0188809,-0.851924],[-1,-1,-1,0],[9E+09,9E+09,9E+09,9E+09,9E+09,9E+09]];
CONST robtarget LHP_035:=[[699.02,379.91,-168.70],[0.497729,-0.043976,0.0365454,-0.865446],[-1,-1,-1,0],[9E+09,9E+09,9E+09,9E+09,9E+09,9E+09]];
CONST robtarget LHP_040:=[[787.77,733.63,-260.02],[0.443404,-0.023228,0.047816,-0.894744],[-1,-1,-1,0],[9E+09,9E+09,9E+09,9E+09,9E+09,9E+09]];
CONST robtarget LHP_045:=[[1033.71,1080.25,-461.77],[0.269846,0.0608739,0.0794631,-0.957686],[-1,-1,0,0],[9E+09,9E+09,9E+09,9E+09,9E+09,9E+09]];
CONST robtarget LHP_050:=[[1247.344,1214.964,-268.134],[0.1820915,0.09153603,0.12369742,-0.97116566],[-1,-1,0,0],[9E9,9E9,9E9,9E9,9E9,9E9]];
CONST robtarget LHP_055:=[[1444.06,1061.60,-239.72],[0.299937,0.0825452,0.0973258,-0.945384],[-1,-1,0,0],[9E+09,9E+09,9E+09,9E+09,9E+09,9E+09]];
CONST robtarget LHP_060:=[[1299.17,382.16,-44.15],[0.616859,0.0635803,0.0620975,-0.78204],[-1,-1,-1,0],[9E+09,9E+09,9E+09,9E+09,9E+09,9E+09]];
CONST robtarget LHP_065:=[[1300.31,401.52,-167.56],[0.611239,0.0803897,0.0809307,-0.783182],[-1,-1,-1,0],[9E+09,9E+09,9E+09,9E+09,9E+09,9E+09]];
CONST robtarget LHP_066:=[[1001.90,512.66,-24.97],[0.296786,-0.0658732,0.0437859,-0.951663],[-1,-1,0,0],[9E+09,9E+09,9E+09,9E+09,9E+09,9E+09]];
CONST robtarget LHP_070:=[[793.037,542.023,-179.693],[0.20754133,0.019031575,0.0932444,-0.9735861],[-1,-1,0,0],[9E9,9E9,9E9,9E9,9E9,9E9]];
CONST robtarget LHP_075:=[[1029.49,400.421,-202.979],[0.39562756,-0.007666591,0.14027788,-0.9076024],[-1,-1,0,0],[9E9,9E9,9E9,9E9,9E9,9E9]];
CONST robtarget LHP_076:=[[1003.66,410.71,-25.68],[0.364211,-0.0883488,0.0244107,-0.926795],[-1,-1,0,0],[9E+09,9E+09,9E+09,9E+09,9E+09,9E+09]];
CONST robtarget LHP_080:=[[1076.251,387.732,-208.342],[0.43962634,0.059819497,0.10055306,-0.8905276],[-1,-1,0,0],[9E9,9E9,9E9,9E9,9E9,9E9]];
CONST robtarget LHP_085:=[[1115.20,414.51,-186.17],[0.4653,0.0650512,0.093708,-0.877772],[-1,-1,-1,0],[9E+09,9E+09,9E+09,9E+09,9E+09,9E+09]];
CONST robtarget LHP_090:=[[1309.91,408.20,-170.92],[0.623524,0.0686372,0.0633877,-0.776202],[-1,-1,-1,0],[9E+09,9E+09,9E+09,9E+09,9E+09,9E+09]];
CONST robtarget LHP_095:=[[1076.52,400.40,-154.53],[0.364233,-0.00446918,0.0919739,-0.926744],[-1,-1,0,0],[9E+09,9E+09,9E+09,9E+09,9E+09,9E+09]];
CONST robtarget LHP_100:=[[1310.60,637.82,-270.26],[0.359347,0.128527,0.122572,-0.916148],[-1,-1,0,0],[9E+09,9E+09,9E+09,9E+09,9E+09,9E+09]];
CONST robtarget LHP_105:=[[1460.75,765.25,-199.93],[0.413853,0.0959722,0.0635622,-0.903036],[-1,-1,0,0],[9E+09,9E+09,9E+09,9E+09,9E+09,9E+09]];
CONST robtarget LHP_110:=[[1503.17,367.15,-201.31],[0.556665,-0.00361148,-0.00229809,-0.830726],[-1,0,-1,0],[9E+09,9E+09,9E+09,9E+09,9E+09,9E+09]];
CONST robtarget LHP_115:=[[1501.83,111.873,-126.486],[0.4980785,0.07501504,0.043025382,-0.862809],[-1,-1,-1,0],[9E9,9E9,9E9,9E9,9E9,9E9]];
CONST robtarget LHP_120:=[[1609.89,158.05,-114.28],[0.588479,0.00198542,0.0011568,-0.808509],[-1,-1,-1,0],[9E+09,9E+09,9E+09,9E+09,9E+09,9E+09]];
CONST robtarget LHP_125:=[[1638.455,381.7,-207.24],[0.5479616,0.037808824,0.05486916,-0.8338453],[-1,-1,-1,0],[9E9,9E9,9E9,9E9,9E9,9E9]];
CONST robtarget LHP_130:=[[1803.59,658.60,-169.61],[0.558229,0.00244183,0.0115732,-0.829603],[-1,-1,-1,0],[9E+09,9E+09,9E+09,9E+09,9E+09,9E+09]];
CONST robtarget LHP_135:=[[1832.913,607.552,669.677],[0.6102957,-0.087358184,0.105843775,-0.78019536],[-1,-1,-1,0],[9E9,9E9,9E9,9E9,9E9,9E9]];
CONST robtarget LHP_140:=[[2270.294,637.607,1817.373],[0.6669749,-0.3265057,0.039168768,-0.6685838],[-1,-1,-1,0],[9E9,9E9,9E9,9E9,9E9,9E9]];

!****************************************************
!* Unterprogramm  : swp_213500_0_st1606_1           *
!* Modell/Typ     : FHS T3,5 R3 (4325mm)            *
!* Applikation    : Punktschweissen Zange 1         *
!* Anlagen/Station: Linie 16 / St1606               *
!* Robotername    : 1606R04                         *
!* Originalautor  : COMAU                           *
!* Erstelldatum   : 28.02.2006                      *
!****************************************************
!*               Aktualisierungen                   *
!*             ====================                 *
!* Datum       : 13.01.2017                         *
!* dz?nderung    : VS30 - Winter PU 2016/17           *
!* Gedz?ndert von: R. Ddz?rrbeck (ese-robotics fdz?r FFT) *
!****************************************************

 INIT_SW_BASE;

 WKZ_1_AUFNEHMEN;

 MoveJ ToolHome1,vSchnell,fine,nomtcp1;


 MoveJ LHP_000,vSchnell,fine,nomtcp1\WObj:=BS_1606_1A;
 Vorhub\auf;

 KOLLISION_ZONE 5\Anfrage;

 ! Warte auf Freigabe SPS, Fahrzeug in Position
 ABL 2\ABL_WAIT;
 ABL 10\ABL_SET;

 KOLLISION_ZONE 1\Anfrage;
 KOLLISION_ZONE 2\Anfrage;
 KOLLISION_ZONE 6\Anfrage;

 MoveJ LHP_005,vSchnell,z100,nomtcp1\WObj:=BS_1606_1A;
 MoveJ LHP_010,vSchnell,z100,nomtcp1\WObj:=BS_1606_1A;
 MoveJ LHP_015,vSchnell,z100,nomtcp1\WObj:=BS_1606_1A;
 MoveJ LHP_020,vSchnell,z100,nomtcp1\WObj:=BS_1606_1A;

 SpotL G0216047007BP20\VFO:=210,vSpot,nomtcp1\WObj:=BS_1606_1A;
 !opt max frueh
 KOLLISION_ZONE 1\Freigabe;

!SWP neue Koordinaden

 SpotL G0216020172BP20\VFO:=210,vSpot,nomtcp1\WObj:=BS_1606_1A;
 !
 !opt norm
 !MoveL G0216020170BP20, vSchnell, fine, nomtcp1\WObj:=BS_1606_1A;
 !KOLLISION_ZONE 1\Freigabe;

 SpotL G0216020170BP20\VFO:=210\Vorhub_Auf,vSpot,nomtcp1\WObj:=BS_1606_1A;

 MoveJ LHP_035,vSchnell,z100,nomtcp1\WObj:=BS_1606_1A;
 MoveJ LHP_040,vSchnell,z100,nomtcp1\WObj:=BS_1606_1A;
 !opt spaet
 !KOLLISION_ZONE 1\Freigabe;
 !
 MoveJ LHP_045,vSchnell,z100,nomtcp1\WObj:=BS_1606_1A;
 !Start Kollision mit Vorrichtung ! (Folie55)
 MoveJ LHP_055,vSchnell,z100,nomtcp1\WObj:=BS_1606_1A;
 !
 !versch
 !
 MoveJ LHP_155, vSchnell, z100, nomtcp1\WObj:=BS_1606_1A;
 MoveJ LHP_145, vSchnell, z80, nomtcp1\WObj:=BS_1606_1A;
 MoveJ LHP_175, vSchnell, z20, nomtcp1\WObj:=BS_1606_1A;
!
! ZMIANA !!!!!
!
WaitUntil FALSE;
 !SpotL G0216020180BP20\VFO:=210\Vorhub_Auf,vSpot,nomtcp1\WObj:=BS_1606_1A;

 !
 MoveL LHP_060, vSchnell, z20, nomtcp1\WObj:=BS_1606_1A;
 MoveJ LHP_065, vSchnell, z50, nomtcp1\WObj:=BS_1606_1A;
 MoveJ LHP_165, vSchnell, z100, nomtcp1\WObj:=BS_1606_1A;
 !Ende Kollision mit Vorrichtung ! (Folie55)
 !ende Versch
 !opt max frueh
 !MoveL G0216020160BP20, vSchnell, fine, nomtcp1\WObj:=BS_1606_1A;
 !KOLLISION_ZONE 2\Freigabe;

 SpotL G0216020160BP20\VFO:=210,vSpot,nomtcp1\WObj:=BS_1606_1A;
 !
 KOLLISION_ZONE 2\Freigabe;

 !alt_Z1\Frei;

 SpotL G0216020158BP20\VFO:=210,vSpot,nomtcp1\WObj:=BS_1606_1A;

 MoveL LHP_066,vSpot,z1,nomtcp1\WObj:=BS_1606_1A;
 MoveL [[1001.89,531.58,-24.98],[0.296786,-0.0658745,0.0437906,-0.951662],[-1,-1,0,0],[9E+09,9E+09,9E+09,9E+09,9E+09,9E+09]], vSpot, z1, nomtcp1\WObj:=BS_1606_1A;
 MoveL [[888.43,535.56,-4.02],[0.256121,-0.0829008,0.0580729,-0.961331],[-1,-1,0,0],[9E+09,9E+09,9E+09,9E+09,9E+09,9E+09]], vSpot, z1, nomtcp1\WObj:=BS_1606_1A;

 SpotL G0216020154BP20\VFO:=210,vSpot,nomtcp1\WObj:=BS_1606_1A;
 !opt spaet
 !KOLLISION_ZONE 2\Freigabe;

 SpotL G0216020152BP20\VFO:=210,vSpot,nomtcp1\WObj:=BS_1606_1A;

 SpotL G0216020150BP20\VFO:=210,vSpot,nomtcp1\WObj:=BS_1606_1A;
 MoveL [[818.08,527.26,7.39],[0.226547,-0.0825521,0.0527165,-0.969063],[-1,-1,0,0],[9E+09,9E+09,9E+09,9E+09,9E+09,9E+09]], vSpot, z1, nomtcp1\WObj:=BS_1606_1A;
 MoveL [[762.43,524.68,12.54],[0.205865,-0.0816334,0.0516716,-0.9738],[-1,-1,0,0],[9E+09,9E+09,9E+09,9E+09,9E+09,9E+09]], vSpot, z1, nomtcp1\WObj:=BS_1606_1A;

 SpotL G0216047004BP20\VFO:=210\Vorhub_Auf,vSpot,nomtcp1\WObj:=BS_1606_1A;

 MoveJ LHP_070,vSchnell,z100,nomtcp1\WObj:=BS_1606_1A;
 MoveJ LHP_075,vSchnell,z100,nomtcp1\WObj:=BS_1606_1A;

 SpotL G0216020168BP20\VFO:=210,vSpot,nomtcp1\WObj:=BS_1606_1A;

 MoveL LHP_076,vSpot,z1,nomtcp1\WObj:=BS_1606_1A;

 SpotL G0216020164BP20\VFO:=210,vSpot,nomtcp1\WObj:=BS_1606_1A;


 SpotL G0216020162BP20\VFO:=210\Vorhub_Auf,vSpot,nomtcp1\WObj:=BS_1606_1A;



 MoveJ LHP_095, vSchnell, z80, nomtcp1\WObj:=BS_1606_1A;
 MoveJ LHP_100,vSchnell,z100,nomtcp1\WObj:=BS_1606_1A;
 MoveJ LHP_105,vSchnell,z100,nomtcp1\WObj:=BS_1606_1A;
 MoveJ LHP_110,vSchnell,z100,nomtcp1\WObj:=BS_1606_1A;

 SpotL G0216021052BP20\VFO:=210,vSpot,nomtcp1\WObj:=BS_1606_1A;


 SpotL G0216021054BP20\VFO:=210,vSpot,nomtcp1\WObj:=BS_1606_1A;
 SpotL G0216021056BP20\VFO:=210,vSpot,nomtcp1\WObj:=BS_1606_1A;
 SpotL G0216021058BP20\VFO:=210,vSpot,nomtcp1\WObj:=BS_1606_1A;
 SpotL G0216021060BP20\VFO:=210\Vorhub_Auf,vSpot,nomtcp1\WObj:=BS_1606_1A;

 MoveJ LHP_115,vSchnell,z100,nomtcp1\WObj:=BS_1606_1A;


 MoveJ LHP_120,vSchnell,z100,nomtcp1\WObj:=BS_1606_1A;

 SpotL G0216021068BP20\VFO:=210,vSpot,nomtcp1\WObj:=BS_1606_1A;

 SpotL G0216021070BP20\VFO:=210,vSpot,nomtcp1\WObj:=BS_1606_1A;

 SpotL G0216021072BP20\VFO:=210\Vorhub_Auf,vSpot,nomtcp1\WObj:=BS_1606_1A;

 MoveJ LHP_125, vSchnell, z200, nomtcp1\WObj:=BS_1606_1A;
 MoveJ LHP_130, vSchnell, fine, nomtcp1\WObj:=BS_1606_1A;
 !alt_Z2\Frei;
 KOLLISION_ZONE 5\Freigabe;
 MoveJ [[1890.64,724.73,327.69],[0.573803,-0.0241173,0.0161225,-0.818479],[-1,-1,-1,0],[9E+09,9E+09,9E+09,9E+09,9E+09,9E+09]], vSchnell, z100, nomtcp1\WObj:=BS_1606_1A;
 MoveJ [[1878.67,697.76,491.78],[0.548784,-0.0234001,0.00386422,-0.835628],[-1,-1,-1,0],[9E+09,9E+09,9E+09,9E+09,9E+09,9E+09]], vSchnell, z100, nomtcp1\WObj:=BS_1606_1A;
 MoveJ [[1918.47,774.29,837.58],[0.611382,0.029609,0.0513063,-0.789116],[-1,-1,-1,0],[9E+09,9E+09,9E+09,9E+09,9E+09,9E+09]], vSchnell, z100, nomtcp1\WObj:=BS_1606_1A;
 MoveJ LHP_140,vSchnell,z100,nomtcp1\WObj:=BS_1606_1A;

 MoveJ ToolHome1,vSchnell,fine,nomtcp1;

 !alt_Z 5\Frei;
 KOLLISION_ZONE 6\Freigabe;

  ! Warte auf Freigabe SPS, Fertigmeldung Schweissen
 ABL 254\ABL_WAIT;
 ABL 255\ABL_SET;

ENDPROC !Punktschweissen Zange 1, FHS T3,5 R3 (4325mm)


PROC swp_215300_0_st1606_1()

CONST robtarget LHP_000:=[[2573.52808,1238.19995,2660.84009],[0.56645757,-0.58473384,0.19941168,-0.54538715],[-1,-1,-1,4],[9E9,9E9,9E9,9E9,9E9,9E9]];
CONST robtarget LHP_005:=[[1360.172,1026.896,440.838989],[0.5866833,0.005191112,0.051883798,-0.80813605],[-1,-1,-1,0],[9E9,9E9,9E9,9E9,9E9,9E9]];
CONST robtarget LHP_010:=[[1032.36804,977.945984,-459.062988],[0.43703678,0.12694271,0.09414318,-0.8854499],[-1,-1,-1,0],[9E9,9E9,9E9,9E9,9E9,9E9]];
CONST robtarget LHP_015:=[[798.565002,757.20697,-251.078003],[0.47486252,-0.019805102,0.048932664,-0.87847537],[-1,-1,-1,0],[9E9,9E9,9E9,9E9,9E9,9E9]];
CONST robtarget LHP_020:=[[687.611023,377.389008,-182.513],[0.5033828,-0.04139257,0.03810638,-0.8622299],[-1,-1,-1,0],[9E9,9E9,9E9,9E9,9E9,9E9]];
CONST robtarget LHP_025:=[[699.05,379.90,-168.79],[0.497735,-0.0439583,0.0365477,-0.865443],[-1,-1,-1,0],[9E+09,9E+09,9E+09,9E+09,9E+09,9E+09]];
CONST robtarget LHP_030:=[[788.08,733.39,-256.84],[0.443411,-0.0232196,0.0478196,-0.89474],[-1,-1,-1,0],[9E+09,9E+09,9E+09,9E+09,9E+09,9E+09]];
CONST robtarget LHP_035:=[[1033.71,1080.19,-461.81],[0.269848,0.0608723,0.0794594,-0.957686],[-1,-1,0,0],[9E+09,9E+09,9E+09,9E+09,9E+09,9E+09]];
CONST robtarget LHP_040:=[[1444.11,1061.50,-239.82],[0.299947,0.0825549,0.0973232,-0.945381],[-1,-1,0,0],[9E+09,9E+09,9E+09,9E+09,9E+09,9E+09]];
CONST robtarget LHP_045:=[[1382.57,676.16,-177.79],[0.528176,0.00137494,0.0696186,-0.846275],[-1,-1,-1,0],[9E+09,9E+09,9E+09,9E+09,9E+09,9E+09]];
CONST robtarget LHP_050:=[[1309.88,408.12,-170.83],[0.616293,0.0691903,0.0627507,-0.781958],[-1,-1,-1,0],[9E+09,9E+09,9E+09,9E+09,9E+09,9E+09]];
CONST robtarget LHP_055:=[[1299.16,382.10,-44.10],[0.616865,0.0635557,0.0620999,-0.782037],[-1,-1,-1,0],[9E+09,9E+09,9E+09,9E+09,9E+09,9E+09]];
CONST robtarget LHP_060:=[[1300.31,401.48,-167.59],[0.611243,0.0803831,0.0809307,-0.78318],[-1,-1,-1,0],[9E+09,9E+09,9E+09,9E+09,9E+09,9E+09]];
CONST robtarget LHP_065:=[[1054.33,541.70,-228.26],[0.365991,0.0660923,0.0753214,-0.925208],[-1,-1,0,0],[9E+09,9E+09,9E+09,9E+09,9E+09,9E+09]];
CONST robtarget LHP_066:=[[1001.86,513.52,-32.15],[0.273973,-0.0669015,0.0422098,-0.958479],[-1,-1,0,0],[9E+09,9E+09,9E+09,9E+09,9E+09,9E+09]];
CONST robtarget LHP_070:=[[976.25,512.62,-27.09],[0.265297,-0.0731468,0.0350815,-0.960748],[-1,-1,0,0],[9E+09,9E+09,9E+09,9E+09,9E+09,9E+09]];
CONST robtarget LHP_075:=[[793.03,542.01,-179.71],[0.195219,0.017852,0.0934789,-0.976131],[-1,-1,0,0],[9E+09,9E+09,9E+09,9E+09,9E+09,9E+09]];
CONST robtarget LHP_080:=[[1036.10,391.37,-206.29],[0.367004,-0.0120429,0.139982,-0.919548],[-1,-1,0,0],[9E+09,9E+09,9E+09,9E+09,9E+09,9E+09]];
CONST robtarget LHP_081:=[[1000.78,413.95,-31.69],[0.375336,-0.0880264,0.0254868,-0.922347],[-1,-1,0,0],[9E+09,9E+09,9E+09,9E+09,9E+09,9E+09]];
CONST robtarget LHP_085:=[[1095.55,389.92,-147.05],[0.364243,-0.00445865,0.0919851,-0.926739],[-1,-1,0,0],[9E+09,9E+09,9E+09,9E+09,9E+09,9E+09]];
CONST robtarget LHP_090:=[[1237.80,591.89,-241.44],[0.358818,0.101999,0.118758,-0.920186],[-1,-1,0,0],[9E+09,9E+09,9E+09,9E+09,9E+09,9E+09]];
CONST robtarget LHP_095:=[[1489.53,806.77,-347.16],[0.411235,0.12926,0.0787946,-0.898871],[-1,-1,0,0],[9E+09,9E+09,9E+09,9E+09,9E+09,9E+09]];
CONST robtarget LHP_100:=[[1890.66,724.71,327.67],[0.573807,-0.0241158,0.016124,-0.818476],[-1,-1,-1,0],[9E+09,9E+09,9E+09,9E+09,9E+09,9E+09]];
CONST robtarget LHP_105:=[[1878.71,697.75,491.71],[0.548792,-0.0233886,0.00387377,-0.835622],[-1,-1,-1,0],[9E+09,9E+09,9E+09,9E+09,9E+09,9E+09]];
CONST robtarget LHP_110:=[[1918.45,774.29,837.58],[0.611379,0.0296046,0.05131,-0.789118],[-1,-1,-1,0],[9E+09,9E+09,9E+09,9E+09,9E+09,9E+09]];
CONST robtarget LHP_115:=[[2270.27,637.61,1817.33],[0.666976,-0.326499,0.0391784,-0.668586],[-1,-1,-1,0],[9E+09,9E+09,9E+09,9E+09,9E+09,9E+09]];

  ! ------------------------------------------------------------
  ! Unterprogramm:
  ! Stand
  ! Daimler AG - Werk Ludwigsfelde
  ! ------------------------------------------------------------
  ! ************************************************************
  ! Kommentar: Achtung
  !            automatisch generiert!!!!!!!!!!!!!!!!!!
  ! ************************************************************

! Robotername:            1606R04
! Anlagenbezeichn:        Linie 16          Stations-Nr:  1606
! Stand / Version:        29.07.2009 / 1.1
! Name Bearbeiter:        Karmann
! Applikationssteuerung:  Punktschweissen
! Baumuster:              FHS T2 R2
! abgedz?ndert, Vorlage 113500

INIT_SW_BASE;

WKZ_1_AUFNEHMEN;

MoveJ ToolHome1,vSchnell,fine,nomtcp1;


MoveJ LHP_000,vSchnell,fine,nomtcp1\WObj:=BS_1606_1A;
Vorhub\auf;

KOLLISION_ZONE 1\Anfrage;

KOLLISION_ZONE 2\Anfrage;

KOLLISION_ZONE 5\Anfrage;

KOLLISION_ZONE 6\Anfrage;

MoveJ LHP_005,vSchnell,z100,nomtcp1\WObj:=BS_1606_1A;
MoveJ LHP_010,vSchnell,z100,nomtcp1\WObj:=BS_1606_1A;
MoveJ LHP_015,vSchnell,z100,nomtcp1\WObj:=BS_1606_1A;
MoveJ LHP_020,vSchnell,z100,nomtcp1\WObj:=BS_1606_1A;

SpotL G0216047007BP20\VFO:=220,vSpot,nomtcp1\WObj:=BS_1606_1A;
MoveL [[788.56,413.18,0.00],[0.583519,-0.0826067,0.0236779,-0.80754],[-1,-1,-1,0],[9E+09,9E+09,9E+09,9E+09,9E+09,9E+09]], vSpot, z10, nomtcp1\WObj:=BS_1606_1A;


SpotL G0216020172BP20\VFO:=220,vSpot,nomtcp1\WObj:=BS_1606_1A;
!
MoveJ G0216020170BP20,vSchnell,fine,nomtcp1\WObj:=BS_1606_1A;
!
KOLLISION_ZONE 1\Freigabe;

SpotL G0216020170BP20\VFO:=220\Vorhub_Auf,vSpot,nomtcp1\WObj:=BS_1606_1A;

MoveJ LHP_025,vSchnell ,z50,nomtcp1\WObj:=BS_1606_1A;

MoveJ LHP_030,vSchnell,z100,nomtcp1\WObj:=BS_1606_1A;
MoveJ LHP_035,vSchnell,z100,nomtcp1\WObj:=BS_1606_1A;
MoveJ LHP_040,vSchnell,z100,nomtcp1\WObj:=BS_1606_1A;
MoveJ LHP_045,vSchnell,z100,nomtcp1\WObj:=BS_1606_1A;
MoveJ LHP_050,vSchnell,z80,nomtcp1\WObj:=BS_1606_1A;
MoveJ [[1299.24,382.13,-44.21],[0.616872,0.0635889,0.0621053,-0.782028],[-1,-1,-1,0],[9E+09,9E+09,9E+09,9E+09,9E+09,9E+09]], vSchnell, z20, nomtcp1\WObj:=BS_1606_1A;
!
! ZMIANA !!!!
!
WaitUntil FALSE;
!SpotL G0216020180BP20\VFO:=210\Vorhub_Auf,vSpot,nomtcp1\WObj:=BS_1606_1A;

MoveL LHP_055,vSchnell,z20,nomtcp1\WObj:=BS_1606_1A;
MoveJ LHP_060,vSchnell,z50,nomtcp1\WObj:=BS_1606_1A;
MoveJ LHP_065,vSchnell,z100,nomtcp1\WObj:=BS_1606_1A;

SpotL G0216020160BP20\VFO:=220,vSpot,nomtcp1\WObj:=BS_1606_1A;

!alt_Z 1\Frei;
KOLLISION_ZONE 2\Freigabe;

SpotL G0216020158BP20\VFO:=220,vSpot,nomtcp1\WObj:=BS_1606_1A;

MoveL LHP_066,vSpot,z1,nomtcp1\WObj:=BS_1606_1A;

MoveJ LHP_070,vSchnell,z100,nomtcp1\WObj:=BS_1606_1A;
MoveL [[976.27,531.40,-18.22],[0.260836,-0.0732981,0.0347512,-0.961969],[-1,-1,0,0],[9E+09,9E+09,9E+09,9E+09,9E+09,9E+09]], vSchnell, z100, nomtcp1\WObj:=BS_1606_1A;
MoveL [[888.42,534.96,-4.05],[0.229574,-0.0844597,0.0557888,-0.968013],[-1,-1,0,0],[9E+09,9E+09,9E+09,9E+09,9E+09,9E+09]], vSchnell, z100, nomtcp1\WObj:=BS_1606_1A;

SpotL G0216020154BP20\VFO:=220,vSpot,nomtcp1\WObj:=BS_1606_1A;

SpotL G0216020152BP20\VFO:=220,vSpot,nomtcp1\WObj:=BS_1606_1A;

SpotL G0216020150BP20\VFO:=220,vSpot,nomtcp1\WObj:=BS_1606_1A;
!
MoveL [[818.05,529.53,-2.20],[0.212761,-0.0832861,0.0515594,-0.972182],[-1,-1,0,0],[9E+09,9E+09,9E+09,9E+09,9E+09,9E+09]], vSchnell, z100, nomtcp1\WObj:=BS_1606_1A;
MoveL [[762.42,528.83,6.44],[0.191518,-0.0823751,0.0504859,-0.976722],[-1,-1,0,0],[9E+09,9E+09,9E+09,9E+09,9E+09,9E+09]], vSchnell, z100, nomtcp1\WObj:=BS_1606_1A;

SpotL G0216047004BP20\VFO:=220\Vorhub_Auf,vSpot,nomtcp1\WObj:=BS_1606_1A;

MoveJ LHP_075,vSchnell,z100,nomtcp1\WObj:=BS_1606_1A;
MoveJ LHP_080,vSchnell,z100,nomtcp1\WObj:=BS_1606_1A;

SpotL G0216020168BP20\VFO:=220,vSpot,nomtcp1\WObj:=BS_1606_1A;

MoveL LHP_081,vSpot,z1,nomtcp1\WObj:=BS_1606_1A;

SpotL G0216020164BP20\VFO:=220,vSpot,nomtcp1\WObj:=BS_1606_1A;


SpotL G0216020162BP20\VFO:=220\Vorhub_Auf,vSpot,nomtcp1\WObj:=BS_1606_1A;

MoveJ LHP_085, vSchnell, z50, nomtcp1\WObj:=BS_1606_1A;
MoveJ LHP_090,vSchnell,z100,nomtcp1\WObj:=BS_1606_1A;
MoveJ LHP_095,vSchnell,z100,nomtcp1\WObj:=BS_1606_1A;
MoveJ LHP_100,vSchnell,z100,nomtcp1\WObj:=BS_1606_1A;
!opt
!KOLLISION_ZONE 5\Freigabe;
MoveJ LHP_105,vSchnell,z100,nomtcp1\WObj:=BS_1606_1A;
MoveJ LHP_110,vSchnell,z100,nomtcp1\WObj:=BS_1606_1A;
MoveJ LHP_115,vSchnell,z100,nomtcp1\WObj:=BS_1606_1A;

MoveJ ToolHome1,vSchnell,fine,nomtcp1;

!alt Z 2\Frei;

KOLLISION_ZONE 5\Freigabe;

ABL 254\ABL_WAIT;

ABL 255\ABL_SET;
!

ENDPROC


PROC swp_215300_0_st1606_1_1()

CONST robtarget LHP_000:=[[2224.893,836.8007,752.8398],[0.75648797,-0.003241744,0.000259822,-0.6539995],[-1,0,-1,0],[9E9,9E9,9E9,9E9,9E9,9E9]];
CONST robtarget LHP_005:=[[1771.084,710.2776,-41.35357],[0.6467643,0.009669394,0.004800967,-0.76261353],[-1,-1,-1,0],[9E9,9E9,9E9,9E9,9E9,9E9]];
CONST robtarget LHP_010:=[[2067.637,719.3843,-46.33118],[0.75679874,0.010297084,0.003249933,-0.6535588],[-1,-1,-1,0],[9E9,9E9,9E9,9E9,9E9,9E9]];
CONST robtarget LHP_015:=[[2224.893,836.8007,752.8398],[0.75648797,-0.003241744,0.000259822,-0.6539995],[-1,0,-1,0],[9E9,9E9,9E9,9E9,9E9,9E9]];

  ! ------------------------------------------------------------
  ! Unterprogramm:
  ! Stand
  ! Daimler AG - Werk Ludwigsfelde
  ! ------------------------------------------------------------
  ! ************************************************************
  ! Kommentar: Achtung
  !            automatisch generiert!!!!!!!!!!!!!!!!!!
  ! ************************************************************

! Robotername:            1606R04
! Anlagenbezeichn:        Linie 16          Stations-Nr:  1606
! Stand / Version:        29.07.2009 / 1.1
! Name Bearbeiter:        Karmann
! Applikationssteuerung:  Punktschweissen
! Baumuster:              FHS T2 R2



INIT_SW_BASE;

WKZ_1_AUFNEHMEN;

MoveJ ToolHome1,vSchnell,fine,nomtcp1;

ABL 2\ABL_WAIT;

ABL 10\ABL_SET;


KOLLISION_ZONE 1\Anfrage;

KOLLISION_ZONE 2\Anfrage;

KOLLISION_ZONE 5\Anfrage;

KOLLISION_ZONE 9\Anfrage;

MoveJ LHP_000,vSchnell,z100,nomtcp1\WObj:=BS_1606_1A;
MoveJ LHP_005,vSchnell,z100,nomtcp1\WObj:=BS_1606_1A;

SpotL G0216022524BP20\VFO:=210,vSpot,nomtcp1\WObj:=BS_1606_1A;

SpotL G0216022526BP20\VFO:=210,vSpot,nomtcp1\WObj:=BS_1606_1A;
SpotL G0216022528BP20\VFO:=210,vSpot,nomtcp1\WObj:=BS_1606_1A;
SpotL G0216022530BP20\VFO:=210,vSpot,nomtcp1\WObj:=BS_1606_1A;
SpotL G0216022532BP20\VFO:=210,vSpot,nomtcp1\WObj:=BS_1606_1A;
SpotL G0216022536BP20\VFO:=210,vSpot,nomtcp1\WObj:=BS_1606_1A;

!SWP entfaellt
!SpotL G0216022538BP20\VFO:=210, vSpot, nomtcp1\WObj:=BS_1606_1A;

SpotL G0216022540BP20\VFO:=210,vSpot,nomtcp1\WObj:=BS_1606_1A;

MoveJ LHP_010,vSchnell,z100,nomtcp1\WObj:=BS_1606_1A;
MoveJ LHP_015,vSchnell,z100,nomtcp1\WObj:=BS_1606_1A;

MoveJ ToolHome1,vSchnell,fine,nomtcp1;

KOLLISION_ZONE 1\Freigabe;

KOLLISION_ZONE 2\Freigabe;

KOLLISION_ZONE 5\Freigabe;

KOLLISION_ZONE 6\Freigabe;

KOLLISION_ZONE 9\Freigabe;

ENDPROC


PROC swp_215500_0_st1606_1()

CONST robtarget LHP_000:=[[2573.52808,1238.19995,2660.84106],[0.56645757,-0.58473384,0.19941168,-0.54538715],[-1,-1,-1,4],[9E9,9E9,9E9,9E9,9E9,9E9]];
CONST robtarget LHP_005:=[[1333.17,1401.02,132.09],[0.584225,0.0885625,0.175362,-0.787455],[-1,-1,-1,0],[9E+09,9E+09,9E+09,9E+09,9E+09,9E+09]];
CONST robtarget LHP_010:=[[987.15,1000.82,-423.48],[0.428568,0.119027,0.092061,-0.890891],[-1,-1,-1,0],[9E+09,9E+09,9E+09,9E+09,9E+09,9E+09]];
CONST robtarget LHP_015:=[[798.56,757.20,-251.08],[0.475639,-0.0318939,0.0359918,-0.878325],[-1,-1,-1,0],[9E+09,9E+09,9E+09,9E+09,9E+09,9E+09]];
CONST robtarget LHP_020:=[[687.611023,377.389008,-182.513],[0.5033828,-0.04139257,0.03810638,-0.8622299],[-1,-1,-1,0],[9E9,9E9,9E9,9E9,9E9,9E9]];
CONST robtarget LHP_025:=[[699.05,379.91,-168.78],[0.497734,-0.0439604,0.0365474,-0.865444],[-1,-1,-1,0],[9E+09,9E+09,9E+09,9E+09,9E+09,9E+09]];
CONST robtarget LHP_030:=[[787.78,733.63,-260.06],[0.443404,-0.0232218,0.0478173,-0.894744],[-1,-1,-1,0],[9E+09,9E+09,9E+09,9E+09,9E+09,9E+09]];
CONST robtarget LHP_035:=[[1033.71,1080.22,-461.80],[0.269846,0.0608736,0.0794606,-0.957686],[-1,-1,0,0],[9E+09,9E+09,9E+09,9E+09,9E+09,9E+09]];
CONST robtarget LHP_040:=[[1444.10,1061.53,-239.80],[0.299945,0.0825541,0.0973255,-0.945381],[-1,-1,0,0],[9E+09,9E+09,9E+09,9E+09,9E+09,9E+09]];
CONST robtarget LHP_045:=[[1382.57,676.17,-177.78],[0.528176,0.00137516,0.0696194,-0.846275],[-1,-1,-1,0],[9E+09,9E+09,9E+09,9E+09,9E+09,9E+09]];
CONST robtarget LHP_050:=[[1309.88,408.13,-170.83],[0.616292,0.0691923,0.0627505,-0.781959],[-1,-1,-1,0],[9E+09,9E+09,9E+09,9E+09,9E+09,9E+09]];
CONST robtarget LHP_055:=[[1299.17,382.14,-44.14],[0.616861,0.0635724,0.0620975,-0.782039],[-1,-1,-1,0],[9E+09,9E+09,9E+09,9E+09,9E+09,9E+09]];
CONST robtarget LHP_060:=[[1300.31,401.50,-167.58],[0.61124,0.0803878,0.0809307,-0.783182],[-1,-1,-1,0],[9E+09,9E+09,9E+09,9E+09,9E+09,9E+09]];
CONST robtarget LHP_065:=[[1054.33,541.72,-228.25],[0.365989,0.0660917,0.0753223,-0.925208],[-1,-1,0,0],[9E+09,9E+09,9E+09,9E+09,9E+09,9E+09]];
CONST robtarget LHP_066:=[[1001.90,512.66,-24.97],[0.296786,-0.0658732,0.0437859,-0.951663],[-1,-1,0,0],[9E+09,9E+09,9E+09,9E+09,9E+09,9E+09]];
CONST robtarget LHP_070:=[[793.036987,542.02301,-179.692993],[0.20754133,0.019031575,0.0932444,-0.9735861],[-1,-1,0,0],[9E9,9E9,9E9,9E9,9E9,9E9]];
CONST robtarget LHP_075:=[[1029.48999,400.42099,-202.979004],[0.39562756,-0.007666591,0.14027788,-0.9076024],[-1,-1,0,0],[9E9,9E9,9E9,9E9,9E9,9E9]];
CONST robtarget LHP_076:=[[1000.84,410.38,-25.24],[0.37926,-0.08793,0.0258433,-0.92074],[-1,-1,0,0],[9E+09,9E+09,9E+09,9E+09,9E+09,9E+09]];
CONST robtarget LHP_080:=[[1095.55,389.94,-147.03],[0.364241,-0.00445932,0.0919839,-0.92674],[-1,-1,0,0],[9E+09,9E+09,9E+09,9E+09,9E+09,9E+09]];
CONST robtarget LHP_085:=[[1237.79,591.91,-241.43],[0.358816,0.102,0.118759,-0.920187],[-1,-1,0,0],[9E+09,9E+09,9E+09,9E+09,9E+09,9E+09]];
CONST robtarget LHP_090:=[[1489.52,806.80,-347.16],[0.411232,0.129262,0.0787982,-0.898872],[-1,-1,0,0],[9E+09,9E+09,9E+09,9E+09,9E+09,9E+09]];
CONST robtarget LHP_095:=[[1469.23,418.79,-181.80],[0.506098,0.0220046,-0.0157458,-0.862051],[-1,0,-1,0],[9E+09,9E+09,9E+09,9E+09,9E+09,9E+09]];
CONST robtarget LHP_100:=[[1585.75903,868.737976,-184.042999],[0.62958896,-0.001844419,0.002234461,-0.776923],[-1,-1,-1,0],[9E9,9E9,9E9,9E9,9E9,9E9]];
CONST robtarget LHP_105:=[[1499.84204,354.274994,-170.001007],[0.48788625,0.06460596,0.07147147,-0.86757416],[-1,-1,0,0],[9E9,9E9,9E9,9E9,9E9,9E9]];
CONST robtarget LHP_110:=[[1515.698,376.503998,-37.7140007],[0.49196577,0.012122404,-0.003482358,-0.87052315],[-1,0,-1,0],[9E9,9E9,9E9,9E9,9E9,9E9]];
CONST robtarget LHP_115:=[[1497.73401,124.461998,-115.32],[0.49093002,0.05575197,0.031571873,-0.86883986],[-1,0,0,0],[9E9,9E9,9E9,9E9,9E9,9E9]];
CONST robtarget LHP_120:=[[1628.05,149.95,-117.00],[0.576442,0.0470283,0.0371016,-0.81494],[-1,-1,-1,0],[9E+09,9E+09,9E+09,9E+09,9E+09,9E+09]];
CONST robtarget LHP_125:=[[1638.46,381.68,-207.25],[0.547963,0.0378083,0.0548674,-0.833844],[-1,-1,-1,0],[9E+09,9E+09,9E+09,9E+09,9E+09,9E+09]];
CONST robtarget LHP_130:=[[1803.59,658.58,-169.61],[0.55823,0.00244128,0.01157,-0.829602],[-1,-1,-1,0],[9E+09,9E+09,9E+09,9E+09,9E+09,9E+09]];
CONST robtarget LHP_135:=[[1890.65,724.72,327.68],[0.573805,-0.0241161,0.0161232,-0.818478],[-1,-1,-1,0],[9E+09,9E+09,9E+09,9E+09,9E+09,9E+09]];
CONST robtarget LHP_140:=[[2270.28,637.61,1817.35],[0.666975,-0.326502,0.0391731,-0.668585],[-1,-1,-1,0],[9E+09,9E+09,9E+09,9E+09,9E+09,9E+09]];

  ! ------------------------------------------------------------
  ! Unterprogramm:
  ! Stand
  ! Daimler AG - Werk Ludwigsfelde
  ! ------------------------------------------------------------
  ! ************************************************************
  ! Kommentar: Achtung
  !            automatisch generiert!!!!!!!!!!!!!!!!!!
  ! ************************************************************

! Robotername:            1606R04
! Anlagenbezeichn:        Linie 16          Stations-Nr:  1606
! Stand / Version:        29.07.2009 / 1.1
! Name Bearbeiter:        Karmann
! Applikationssteuerung:  Punktschweissen
! Baumuster:              FHS T2 R3
! abgedz?ndert, Vorlage 113500

INIT_SW_BASE;

WKZ_1_AUFNEHMEN;

MoveJ ToolHome1,vSchnell,fine,nomtcp1;


MoveJ LHP_000,vSchnell,fine,nomtcp1\WObj:=BS_1606_1A;
Vorhub\auf;

KOLLISION_ZONE 1\Anfrage;

KOLLISION_ZONE 2\Anfrage;

KOLLISION_ZONE 5\Anfrage;

KOLLISION_ZONE 6\Anfrage;


MoveJ LHP_005,vSchnell,z100,nomtcp1\WObj:=BS_1606_1A;
MoveJ LHP_010,vSchnell,z100,nomtcp1\WObj:=BS_1606_1A;
MoveJ LHP_015,vSchnell,z100,nomtcp1\WObj:=BS_1606_1A;
MoveJ LHP_020,vSchnell,z100,nomtcp1\WObj:=BS_1606_1A;

SpotL G0216047007BP20\VFO:=220,vSpot,nomtcp1\WObj:=BS_1606_1A;
 !opt max frueh
 !KOLLISION_ZONE 1\Freigabe;


SpotL G0216020172BP20\VFO:=220,vSpot,nomtcp1\WObj:=BS_1606_1A;
!
MoveJ G0216020170BP20, vSchnell, fine, nomtcp1\WObj:=BS_1606_1A;
 !opt max spaet
 KOLLISION_ZONE 1\Freigabe;

SpotL G0216020170BP20\VFO:=220\Vorhub_Auf,vSpot,nomtcp1\WObj:=BS_1606_1A;

MoveJ LHP_025,vSchnell ,z100,nomtcp1\WObj:=BS_1606_1A;

MoveJ LHP_030,vSchnell,z100,nomtcp1\WObj:=BS_1606_1A;
MoveJ LHP_035,vSchnell,z100,nomtcp1\WObj:=BS_1606_1A;
MoveJ LHP_040,vSchnell,z100,nomtcp1\WObj:=BS_1606_1A;
MoveJ LHP_045,vSchnell,z100,nomtcp1\WObj:=BS_1606_1A;
MoveJ LHP_050,vSchnell,z80,nomtcp1\WObj:=BS_1606_1A;
!verschieb
 MoveJ [[1299.24,382.13,-44.21],[0.616872,0.0635889,0.0621053,-0.782028],[-1,-1,-1,0],[9E+09,9E+09,9E+09,9E+09,9E+09,9E+09]], vSchnell, z20, nomtcp1\WObj:=BS_1606_1A;
!
! ZMIANA !!!!
!
WaitUntil FALSE;
!SpotL G0216020180BP20\VFO:=210\Vorhub_Auf,vSpot,nomtcp1\WObj:=BS_1606_1A;

MoveL LHP_055,vSchnell,z20,nomtcp1\WObj:=BS_1606_1A;
MoveJ LHP_060,vSchnell,z50,nomtcp1\WObj:=BS_1606_1A;
MoveJ LHP_065,vSchnell,z100,nomtcp1\WObj:=BS_1606_1A;

SpotL G0216020160BP20\VFO:=220,vSpot,nomtcp1\WObj:=BS_1606_1A;

!altZ 1\Frei;
KOLLISION_ZONE 2\Freigabe;

SpotL G0216020158BP20\VFO:=220,vSpot,nomtcp1\WObj:=BS_1606_1A;

MoveL LHP_066,vSpot,z1,nomtcp1\WObj:=BS_1606_1A;

SpotL G0216020154BP20\VFO:=220,vSpot,nomtcp1\WObj:=BS_1606_1A;

SpotL G0216020152BP20\VFO:=220,vSpot,nomtcp1\WObj:=BS_1606_1A;

SpotL G0216020150BP20\VFO:=220,vSpot,nomtcp1\WObj:=BS_1606_1A;
!
MoveL [[818.05,526.78,7.38],[0.21338,-0.08326,0.0516028,-0.972046],[-1,-1,0,0],[9E+09,9E+09,9E+09,9E+09,9E+09,9E+09]], vSpot, z1, nomtcp1\WObj:=BS_1606_1A;
MoveL [[762.45,526.18,12.53],[0.197611,-0.0820702,0.0509916,-0.975507],[-1,-1,0,0],[9E+09,9E+09,9E+09,9E+09,9E+09,9E+09]], vSpot, z1, nomtcp1\WObj:=BS_1606_1A;

SpotL G0216047004BP20\VFO:=220\Vorhub_Auf,vSpot,nomtcp1\WObj:=BS_1606_1A;

MoveJ LHP_070,vSchnell,z100,nomtcp1\WObj:=BS_1606_1A;
MoveJ LHP_075,vSchnell,z100,nomtcp1\WObj:=BS_1606_1A;

SpotL G0216020168BP20\VFO:=220,vSpot,nomtcp1\WObj:=BS_1606_1A;

MoveL LHP_076,vSpot,z1,nomtcp1\WObj:=BS_1606_1A;

SpotL G0216020164BP20\VFO:=220,vSpot,nomtcp1\WObj:=BS_1606_1A;


SpotL G0216020162BP20\VFO:=220\Vorhub_Auf,vSpot,nomtcp1\WObj:=BS_1606_1A;

MoveJ LHP_080, vSchnell, z50, nomtcp1\WObj:=BS_1606_1A;
MoveJ LHP_085,vSchnell,z100,nomtcp1\WObj:=BS_1606_1A;
MoveJ LHP_090,vSchnell,z100,nomtcp1\WObj:=BS_1606_1A;
MoveJ LHP_095,vSchnell,z100,nomtcp1\WObj:=BS_1606_1A;


SpotL G0216023456BP20\VFO:=210,vSpot,nomtcp1\WObj:=BS_1606_1A;

SpotL G0216023458BP20\VFO:=210,vSpot,nomtcp1\WObj:=BS_1606_1A;

SpotL G0216023460BP20\VFO:=210,vSpot,nomtcp1\WObj:=BS_1606_1A;

SpotL G0216023572BP20\VFO:=210,vSpot,nomtcp1\WObj:=BS_1606_1A;

SpotL G0216023462BP20\VFO:=210\Vorhub_Auf,vSpot,nomtcp1\WObj:=BS_1606_1A;

MoveJ LHP_115,vSchnell,z100,nomtcp1\WObj:=BS_1606_1A;

MoveJ LHP_120,vSchnell,z100,nomtcp1\WObj:=BS_1606_1A;
!4pkt orie

SpotL G0216023468BP20\VFO:=210,vSpot,nomtcp1\WObj:=BS_1606_1A;

SpotL G0216023574BP20\VFO:=210,vSpot,nomtcp1\WObj:=BS_1606_1A;

SpotL G0216023470BP20\VFO:=210,vSpot,nomtcp1\WObj:=BS_1606_1A;

SpotL G0216023472BP20\VFO:=210,vSpot,nomtcp1\WObj:=BS_1606_1A;

SpotL G0216023474BP20\VFO:=210\Vorhub_Auf,vSpot,nomtcp1\WObj:=BS_1606_1A;

MoveJ LHP_125,vSchnell,z100,nomtcp1\WObj:=BS_1606_1A;
MoveJ LHP_130, vSchnell, fine, nomtcp1\WObj:=BS_1606_1A;
!
 KOLLISION_ZONE 5\Freigabe;

MoveJ LHP_135,vSchnell,z100,nomtcp1\WObj:=BS_1606_1A;
MoveJ [[1878.70,697.76,491.72],[0.54879,-0.0233897,0.00387175,-0.835624],[-1,-1,-1,0],[9E+09,9E+09,9E+09,9E+09,9E+09,9E+09]], vSchnell, z100, nomtcp1\WObj:=BS_1606_1A;
MoveJ [[1918.46,774.29,837.58],[0.61138,0.0296061,0.0513081,-0.789117],[-1,-1,-1,0],[9E+09,9E+09,9E+09,9E+09,9E+09,9E+09]], vSchnell, z100, nomtcp1\WObj:=BS_1606_1A;
! alt Z 2\Frei;
MoveJ LHP_140,vSchnell,z100,nomtcp1\WObj:=BS_1606_1A;

MoveJ ToolHome1,vSchnell,fine,nomtcp1;

!alt_Z 5\Frei;

ABL 254\ABL_WAIT;

ABL 255\ABL_SET;

ENDPROC


PROC swp_215500_0_st1606_1_1()

CONST robtarget LHP_000:=[[2298.80908,1087.04395,1641.68396],[0.7011981,-0.2564904,0.02587284,-0.6647289],[-1,0,-1,0],[9E9,9E9,9E9,9E9,9E9,9E9]];
CONST robtarget LHP_005:=[[2067.98193,918.654785,1009.27698],[0.7007552,-0.19723861,-0.035684966,-0.68466467],[-1,0,-1,0],[9E9,9E9,9E9,9E9,9E9,9E9]];
CONST robtarget LHP_010:=[[1788.81299,649.896606,-32.4160805],[0.5975366,-0.010706378,-0.008460994,-0.8017255],[-1,0,-1,0],[9E9,9E9,9E9,9E9,9E9,9E9]];
CONST robtarget LHP_015:=[[1845.44,1048.29,-50.40],[0.704002,0.00758229,0.0070488,-0.710123],[-1,-1,-1,0],[9E+09,9E+09,9E+09,9E+09,9E+09,9E+09]];
CONST robtarget LHP_020:=[[2042.48499,1296.37903,882.351013],[0.7007552,-0.19723861,-0.035684966,-0.68466467],[-1,0,-1,0],[9E9,9E9,9E9,9E9,9E9,9E9]];
CONST robtarget LHP_025:=[[2251.5249,1464.76697,1521.16296],[0.7011981,-0.2564904,0.02587284,-0.6647289],[-1,0,-1,0],[9E9,9E9,9E9,9E9,9E9,9E9]];

  ! ------------------------------------------------------------
  ! Unterprogramm:
  ! Stand
  ! Daimler AG - Werk Ludwigsfelde
  ! ------------------------------------------------------------
  ! ************************************************************
  ! Kommentar: Achtung
  !            automatisch generiert!!!!!!!!!!!!!!!!!!
  ! ************************************************************

! Robotername:            1606R04
! Anlagenbezeichn:        Linie 16          Stations-Nr:  1606
! Stand / Version:        28.07.2009 / 1.3
! Name Bearbeiter:        Karmann
! Applikationssteuerung:  Punktschweissen
! Baumuster:              FHS T2 R3


INIT_SW_BASE;

WKZ_1_AUFNEHMEN;

MoveJ ToolHome1,vSchnell,fine,nomtcp1;


ABL 2\ABL_WAIT;
ABL 10\ABL_SET;


KOLLISION_ZONE 1\Anfrage;

KOLLISION_ZONE 2\Anfrage;

KOLLISION_ZONE 5\Anfrage;

KOLLISION_ZONE 9\Anfrage;

MoveJ LHP_000,vSchnell,z100,nomtcp1\WObj:=BS_1606_1A;
MoveJ LHP_005,vSchnell,z100,nomtcp1\WObj:=BS_1606_1A;

MoveJ LHP_010,vSchnell,fine,nomtcp1\WObj:=BS_1606_1A;

SpotL G0216023226BP20\VFO:=210,vSpot,nomtcp1\WObj:=BS_1606_1A;
SpotL G0216023228BP20\VFO:=210,vSpot,nomtcp1\WObj:=BS_1606_1A;
SpotL G0216023230BP20\VFO:=210,vSpot,nomtcp1\WObj:=BS_1606_1A;
SpotL G0216023232BP20\VFO:=210,vSpot,nomtcp1\WObj:=BS_1606_1A;
SpotL G0216023234BP20\VFO:=210,vSpot,nomtcp1\WObj:=BS_1606_1A;
SpotL G0216023236BP20\VFO:=210,vSpot,nomtcp1\WObj:=BS_1606_1A;
SpotL G0216023238BP20\VFO:=210,vSpot,nomtcp1\WObj:=BS_1606_1A;


SpotL G0216021634BP20\VFO:=210,vSpot,nomtcp1\WObj:=BS_1606_1A;
SpotL G0216023242BP20\VFO:=210,vSpot,nomtcp1\WObj:=BS_1606_1A;
SpotL G0216023244BP20\VFO:=210,vSpot,nomtcp1\WObj:=BS_1606_1A;

MoveJ LHP_015,vSchnell,z100,nomtcp1\WObj:=BS_1606_1A;
MoveJ LHP_020,vSchnell,z100,nomtcp1\WObj:=BS_1606_1A;
MoveJ LHP_025,vSchnell,z100,nomtcp1\WObj:=BS_1606_1A;

MoveJ ToolHome1,vSchnell,fine,nomtcp1;

KOLLISION_ZONE 1\Freigabe;

KOLLISION_ZONE 2\Freigabe;

KOLLISION_ZONE 5\Freigabe;

KOLLISION_ZONE 6\Freigabe;

KOLLISION_ZONE 9\Freigabe;
!

ENDPROC


PROC swp_223100_0_st1606_1()

CONST robtarget LHP_000:=[[2573.53101,1238.19995,2660.84204],[0.56645757,-0.58473384,0.19941168,-0.54538715],[-1,-1,-1,4],[9E9,9E9,9E9,9E9,9E9,9E9]];
CONST robtarget LHP_005:=[[1933.57397,1076.34998,919.023987],[0.6739808,-0.04561597,0.22679393,-0.70159364],[-1,-1,-1,0],[9E9,9E9,9E9,9E9,9E9,9E9]];
CONST robtarget LHP_010:=[[1910.90503,994.687988,216.904999],[0.7042605,0.08468377,0.09847328,-0.6979605],[-1,-1,-1,0],[9E9,9E9,9E9,9E9,9E9,9E9]];
CONST robtarget LHP_015:=[[1910.89099,994.690002,-385.321991],[0.683501,0.087539785,0.09595496,-0.71830064],[-1,-1,-1,0],[9E9,9E9,9E9,9E9,9E9,9E9]];
CONST robtarget LHP_020:=[[1910.92,803.63,-358.65],[0.683496,0.087554,0.0959515,-0.718305],[-1,-1,-1,0],[9E+09,9E+09,9E+09,9E+09,9E+09,9E+09]];
CONST robtarget LHP_025:=[[1910.97,741.50,-281.66],[0.683494,0.0875455,0.0959486,-0.718307],[-1,-1,-1,0],[9E+09,9E+09,9E+09,9E+09,9E+09,9E+09]];
CONST robtarget LHP_030:=[[1910.91,559.83,-213.69],[0.686476,0.0613746,0.0695917,-0.721208],[-1,-1,-1,0],[9E+09,9E+09,9E+09,9E+09,9E+09,9E+09]];
CONST robtarget LHP_035:=[[1929.33,361.88,-170.13],[0.702471,0.0120548,-0.002609,-0.711605],[-1,0,-1,0],[9E+09,9E+09,9E+09,9E+09,9E+09,9E+09]];
CONST robtarget LHP_040:=[[2007.526,383.55899,-50.7519989],[0.75072795,0.000611088,0.00040383,-0.6606111],[-1,-1,-1,0],[9E9,9E9,9E9,9E9,9E9,9E9]];
CONST robtarget LHP_045:=[[1993.04797,313.046997,-31.7070007],[0.7336252,0.009941696,-0.001285905,-0.67948043],[-1,0,-1,0],[9E9,9E9,9E9,9E9,9E9,9E9]];
CONST robtarget LHP_050:=[[2002.59399,189.292999,-35.1940002],[0.73792726,0.009937888,-0.0012356,-0.67480594],[-1,0,-1,0],[9E9,9E9,9E9,9E9,9E9,9E9]];
CONST robtarget LHP_055:=[[1987.44,-5.82,-69.73],[0.747483,0.000551369,0.000433351,-0.664281],[-1,-1,-1,0],[9E+09,9E+09,9E+09,9E+09,9E+09,9E+09]];
CONST robtarget LHP_060:=[[1929.34,361.89,-170.15],[0.70247,0.0120598,-0.00260928,-0.711607],[-1,0,-1,0],[9E+09,9E+09,9E+09,9E+09,9E+09,9E+09]];
CONST robtarget LHP_065:=[[1910.91,559.85,-213.71],[0.686472,0.0613779,0.0695915,-0.721211],[-1,-1,-1,0],[9E+09,9E+09,9E+09,9E+09,9E+09,9E+09]];
CONST robtarget LHP_070:=[[1769.54,626.69,-228.36],[0.648406,0.063605,0.0595836,-0.756289],[-1,-1,-1,0],[9E+09,9E+09,9E+09,9E+09,9E+09,9E+09]];
CONST robtarget LHP_075:=[[1629.23,373.82,-175.88],[0.60566,0.011527,-0.00436593,-0.795628],[-1,0,-1,0],[9E+09,9E+09,9E+09,9E+09,9E+09,9E+09]];
CONST robtarget LHP_080:=[[1643.37,44.45,-93.67],[0.638426,0.0118697,-0.00343011,-0.769584],[-1,0,-1,0],[9E+09,9E+09,9E+09,9E+09,9E+09,9E+09]];
CONST robtarget LHP_085:=[[1645.79,51.65,-47.78],[0.621544,0.019299,-0.00963586,-0.783082],[-1,0,-1,0],[9E+09,9E+09,9E+09,9E+09,9E+09,9E+09]];
CONST robtarget LHP_090:=[[1652.62,133.53,-52.42],[0.605581,0.0130855,-0.00581803,-0.795655],[-1,0,-1,0],[9E+09,9E+09,9E+09,9E+09,9E+09,9E+09]];
CONST robtarget LHP_095:=[[1617.10803,350.912994,-180.268005],[0.56401443,0.037766688,0.053717423,-0.8231499],[-1,-1,-1,0],[9E9,9E9,9E9,9E9,9E9,9E9]];
CONST robtarget LHP_100:=[[1517.84,635.47,-254.71],[0.565141,-0.00404407,-0.00655324,-0.824958],[-1,0,-1,0],[9E+09,9E+09,9E+09,9E+09,9E+09,9E+09]];
CONST robtarget LHP_105:=[[1647.70,917.36,-357.05],[0.686537,0.012902,0.00966857,-0.726916],[-1,-1,-1,0],[9E+09,9E+09,9E+09,9E+09,9E+09,9E+09]];
CONST robtarget LHP_110:=[[1402.01,954.02,-347.18],[0.618002,-0.00350893,0.00682793,-0.786139],[-1,-1,-1,0],[9E+09,9E+09,9E+09,9E+09,9E+09,9E+09]];
CONST robtarget LHP_115:=[[1380.13,800.38,-344.28],[0.663576,-0.00391562,0.00660285,-0.74807],[-1,-1,-1,0],[9E+09,9E+09,9E+09,9E+09,9E+09,9E+09]];
CONST robtarget LHP_120:=[[1355.05,688.92,-230.68],[0.643458,-0.00406434,0.0069742,-0.765439],[-1,-1,-1,0],[9E+09,9E+09,9E+09,9E+09,9E+09,9E+09]];
CONST robtarget LHP_125:=[[1338.98,616.80,-217.15],[0.641931,-0.00377363,0.00673657,-0.766724],[-1,-1,-1,0],[9E+09,9E+09,9E+09,9E+09,9E+09,9E+09]];
CONST robtarget LHP_130:=[[1328.82,551.60,-198.45],[0.643236,-0.00380631,0.00669098,-0.765629],[-1,-1,-1,0],[9E+09,9E+09,9E+09,9E+09,9E+09,9E+09]];
CONST robtarget LHP_135:=[[1301.19,432.03,-200.08],[0.630965,0.0270779,0.0228783,-0.775001],[-1,-1,-1,0],[9E+09,9E+09,9E+09,9E+09,9E+09,9E+09]];
CONST robtarget LHP_140:=[[1315.22,418.75,-159.95],[0.640955,0.052567,0.0459758,-0.764395],[-1,-1,-1,0],[9E+09,9E+09,9E+09,9E+09,9E+09,9E+09]];
CONST robtarget LHP_145:=[[1314.89,402.01,-58.59],[0.643636,0.0406528,0.0359674,-0.763405],[-1,-1,-1,0],[9E+09,9E+09,9E+09,9E+09,9E+09,9E+09]];
CONST robtarget LHP_150:=[[1314.89,402.00,-58.59],[0.64363700,0.04065100,0.0359677,-0.7634040],[-1,-1,-1,0],[9E+09,9E+09,9E+09,9E+09,9E+09,9E+09]];
CONST robtarget LHP_155:=[[1315.25,418.75,-159.98],[0.640959,0.05257270,0.04597540,-0.7643910],[-1,-1,-1,0],[9E+09,9E+09,9E+09,9E+09,9E+09,9E+09]];
CONST robtarget LHP_160:=[[1301.20,432.03,-200.09],[0.630966,0.0270787,0.0228773,-0.775],[-1,-1,-1,0],[9E+09,9E+09,9E+09,9E+09,9E+09,9E+09]];
CONST robtarget LHP_165:=[[1328.84,551.60,-198.48],[0.643767,-0.00379566,0.00669219,-0.765183],[-1,-1,-1,0],[9E+09,9E+09,9E+09,9E+09,9E+09,9E+09]];
CONST robtarget LHP_170:=[[1356.81,663.69,-214.66],[0.64609,-0.00377796,0.00670482,-0.7632220],[-1,-1,-1,0],[9E+09,9E+09,9E+09,9E+09,9E+09,9E+09]];
CONST robtarget LHP_175:=[[1392.11,854.36,-332.56],[0.646087,-0.00378276,0.00670552,-0.763225],[-1,-1,-1,0],[9E+09,9E+09,9E+09,9E+09,9E+09,9E+09]];
CONST robtarget LHP_180:=[[1598.97,792.20,-328.95],[0.645533,-0.00386844,0.00655628,-0.763695],[-1,-1,-1,0],[9E+09,9E+09,9E+09,9E+09,9E+09,9E+09]];
CONST robtarget LHP_185:=[[1639.58,637.50,-242.37],[0.696285,-0.0006598,0.00564053,-0.717743],[-1,-1,-1,0],[9E+09,9E+09,9E+09,9E+09,9E+09,9E+09]];
CONST robtarget LHP_190:=[[1777.10,396.39,-174.51],[0.778298,0.00338922,-0.00251072,-0.62788],[-1,0,-1,0],[9E+09,9E+09,9E+09,9E+09,9E+09,9E+09]];
CONST robtarget LHP_195:=[[1816.72,397.75,-147.92],[0.816486,0.00152322,-0.000785194,-0.577362],[-1,0,-1,0],[9E+09,9E+09,9E+09,9E+09,9E+09,9E+09]];
CONST robtarget LHP_200:=[[1816.69,397.74,-147.92],[0.816487,0.00151316,-0.000780112,-0.577362],[-1,0,-1,0],[9E+09,9E+09,9E+09,9E+09,9E+09,9E+09]];
CONST robtarget LHP_205:=[[1684.96,400.32,-66.05],[0.598236,-0.000466937,-0.0146474,-0.801186],[-1,0,-1,0],[9E+09,9E+09,9E+09,9E+09,9E+09,9E+09]];
CONST robtarget LHP_210:=[[1780.19,416.87,-42.66],[0.652203,0.00240561,0.00350185,-0.758032],[-1,-1,-1,0],[9E+09,9E+09,9E+09,9E+09,9E+09,9E+09]];
CONST robtarget LHP_215:=[[1614.81,303.29,-114.97],[0.595541,4.37463E-06,7.52158E-05,-0.803325],[-1,-1,-1,0],[9E+09,9E+09,9E+09,9E+09,9E+09,9E+09]];
CONST robtarget LHP_220:=[[1496.10,381.00,-140.90],[0.501832,0.0142883,0.0357857,-0.864106],[-1,-1,-1,0],[9E+09,9E+09,9E+09,9E+09,9E+09,9E+09]];
CONST robtarget LHP_225:=[[1496.16,381.04,-179.37],[0.501836,0.0143261,0.0358019,-0.864103],[-1,-1,-1,0],[9E+09,9E+09,9E+09,9E+09,9E+09,9E+09]];
CONST robtarget LHP_230:=[[1517.37,556.59,-186.35],[0.545787,0.0365786,0.0545327,-0.835347],[-1,-1,-1,0],[9E+09,9E+09,9E+09,9E+09,9E+09,9E+09]];
CONST robtarget LHP_235:=[[1517.83105,635.476013,-254.694],[0.56514114,-0.004049276,-0.006550022,-0.8249583],[-1,0,-1,0],[9E9,9E9,9E9,9E9,9E9,9E9]];
CONST robtarget LHP_240:=[[1558.44,796.09,-349.49],[0.583985,0.0684408,0.0319346,-0.808244],[-1,-1,-1,0],[9E+09,9E+09,9E+09,9E+09,9E+09,9E+09]];
CONST robtarget LHP_245:=[[1477.93,985.71,-357.82],[0.551096,0.0897034,0.0519627,-0.827978],[-1,-1,-1,0],[9E+09,9E+09,9E+09,9E+09,9E+09,9E+09]];
CONST robtarget LHP_250:=[[807.86,896.51,-348.98],[0.475989,-0.019585,0.0486327,-0.877887],[-1,-1,-1,0],[9E+09,9E+09,9E+09,9E+09,9E+09,9E+09]];
CONST robtarget LHP_255:=[[807.84,813.89,-348.98],[0.47599,-0.0195894,0.0486332,-0.877887],[-1,-1,-1,0],[9E+09,9E+09,9E+09,9E+09,9E+09,9E+09]];
CONST robtarget LHP_260:=[[798.625,757.187988,-251.093002],[0.47488588,-0.019798715,0.048936285,-0.8784627],[-1,-1,-1,0],[9E9,9E9,9E9,9E9,9E9,9E9]];
CONST robtarget LHP_265:=[[687.672974,377.386993,-182.552002],[0.5034063,-0.04137853,0.03811411,-0.8622165],[-1,-1,-1,0],[9E9,9E9,9E9,9E9,9E9,9E9]];
CONST robtarget LHP_270:=[[796.06,403.61,2.12],[0.54967,-0.0809587,0.0198978,-0.831212],[-1,-1,-1,0],[9E+09,9E+09,9E+09,9E+09,9E+09,9E+09]];
CONST robtarget LHP_275:=[[951.56,404.05,-36.64],[0.666081,-0.0483269,0.018538,-0.744081],[-1,-1,-1,0],[9E+09,9E+09,9E+09,9E+09,9E+09,9E+09]];
CONST robtarget LHP_280:=[[1053.17,384.08,-147.35],[0.741703,0.0276666,0.0554714,-0.667858],[-1,-1,-1,0],[9E+09,9E+09,9E+09,9E+09,9E+09,9E+09]];
CONST robtarget LHP_285:=[[1117.00,437.68,-186.63],[0.764604,0.0628167,0.0737039,-0.637183],[-1,-1,-1,0],[9E+09,9E+09,9E+09,9E+09,9E+09,9E+09]];
CONST robtarget LHP_290:=[[1206.43,437.70,-186.66],[0.808318,0.0679399,0.0690137,-0.580726],[-1,-1,-1,0],[9E+09,9E+09,9E+09,9E+09,9E+09,9E+09]];
CONST robtarget LHP_295:=[[1254.01,306.17,-147.47],[0.819239,0.0692406,0.0677067,-0.565215],[-1,-1,-1,0],[9E+09,9E+09,9E+09,9E+09,9E+09,9E+09]];
CONST robtarget LHP_300:=[[1294.76,251.64,-118.31],[0.839473,0.0657832,0.0563212,-0.536456],[-1,-1,-1,0],[9E+09,9E+09,9E+09,9E+09,9E+09,9E+09]];
CONST robtarget LHP_305:=[[1302.68,268.91,-77.08],[0.850295,0.0194976,0.0312356,-0.525017],[-1,-1,-1,0],[9E+09,9E+09,9E+09,9E+09,9E+09,9E+09]];
CONST robtarget LHP_310:=[[1302.67,268.92,-77.09],[0.850295,0.0194964,0.0312402,-0.525016],[-1,-1,-1,0],[9E+09,9E+09,9E+09,9E+09,9E+09,9E+09]];
CONST robtarget LHP_315:=[[1294.76,251.64,-118.31],[0.839473,0.0657839,0.0563209,-0.536456],[-1,-1,-1,0],[9E+09,9E+09,9E+09,9E+09,9E+09,9E+09]];
CONST robtarget LHP_320:=[[1254.01,306.17,-147.47],[0.819239,0.0692405,0.0677067,-0.565215],[-1,-1,-1,0],[9E+09,9E+09,9E+09,9E+09,9E+09,9E+09]];
CONST robtarget LHP_325:=[[1206.43,437.70,-186.66],[0.808318,0.0679399,0.0690137,-0.580726],[-1,-1,-1,0],[9E+09,9E+09,9E+09,9E+09,9E+09,9E+09]];
CONST robtarget LHP_330:=[[1117.00,437.68,-186.63],[0.764604,0.0628167,0.0737039,-0.637183],[-1,-1,-1,0],[9E+09,9E+09,9E+09,9E+09,9E+09,9E+09]];
CONST robtarget LHP_335:=[[1116.98,404.12,-155.12],[0.767929,0.0632076,0.0733697,-0.633172],[-1,-1,-1,0],[9E+09,9E+09,9E+09,9E+09,9E+09,9E+09]];
CONST robtarget LHP_340:=[[1116.98,404.12,-77.86],[0.763388,0.0288222,0.0341692,-0.644392],[-1,-1,-1,0],[9E+09,9E+09,9E+09,9E+09,9E+09,9E+09]];
CONST robtarget LHP_345:=[[951.56,404.05,-36.63],[0.666079,-0.0483271,0.018537,-0.744083],[-1,-1,-1,0],[9E+09,9E+09,9E+09,9E+09,9E+09,9E+09]];
CONST robtarget LHP_350:=[[863.42,413.34,0.81],[0.590286,-0.0726155,0.0279581,-0.803435],[-1,-1,-1,0],[9E+09,9E+09,9E+09,9E+09,9E+09,9E+09]];
CONST robtarget LHP_355:=[[687.66803,377.371002,-182.531006],[0.5034058,-0.04138605,0.0381097,-0.8622166],[-1,-1,-1,0],[9E9,9E9,9E9,9E9,9E9,9E9]];
CONST robtarget LHP_360:=[[798.580994,757.198975,-251.070007],[0.47486982,-0.019813199,0.04892835,-0.8784715],[-1,-1,-1,0],[9E9,9E9,9E9,9E9,9E9,9E9]];
CONST robtarget LHP_365:=[[961.40,981.11,-456.97],[0.440335,0.0935079,0.0750373,-0.889792],[-1,-1,-1,0],[9E+09,9E+09,9E+09,9E+09,9E+09,9E+09]];
CONST robtarget LHP_370:=[[1477.90,985.72,-357.83],[0.558631,0.0901634,0.0511329,-0.822914],[-1,-1,-1,0],[9E+09,9E+09,9E+09,9E+09,9E+09,9E+09]];
CONST robtarget LHP_375:=[[1538.22,786.86,-339.64],[0.544053,0.0691445,0.0535195,-0.834482],[-1,-1,-1,0],[9E+09,9E+09,9E+09,9E+09,9E+09,9E+09]];
CONST robtarget LHP_380:=[[1502.92,670.32,-266.02],[0.529086,0.0479959,0.0506422,-0.845695],[-1,-1,-1,0],[9E+09,9E+09,9E+09,9E+09,9E+09,9E+09]];
CONST robtarget LHP_385:=[[1496.13,395.81,-167.92],[0.501832,0.0142997,0.0357903,-0.864106],[-1,-1,-1,0],[9E+09,9E+09,9E+09,9E+09,9E+09,9E+09]];
CONST robtarget LHP_390:=[[1515.01,305.29,-41.45],[0.500229,-6.95049E-05,2.93455E-05,-0.865893],[-1,-1,-1,0],[9E+09,9E+09,9E+09,9E+09,9E+09,9E+09]];
CONST robtarget LHP_395:=[[1371.85706,156.694901,-47.4344292],[0.4850808,-0.004593692,-0.00611278,-0.8744359],[-1,0,-1,0],[9E9,9E9,9E9,9E9,9E9,9E9]];
CONST robtarget LHP_400:=[[1371.81006,156.684998,-41.7470016],[0.48507392,-0.004586132,-0.006106427,-0.8744398],[-1,0,-1,0],[9E9,9E9,9E9,9E9,9E9,9E9]];
CONST robtarget LHP_405:=[[1492.72,315.84,-138.22],[0.571745,-0.00395765,-0.00657566,-0.820395],[-1,0,-1,0],[9E+09,9E+09,9E+09,9E+09,9E+09,9E+09]];
CONST robtarget LHP_410:=[[1568.64,542.95,-202.94],[0.571744,-0.00395848,-0.00658119,-0.820396],[-1,0,-1,0],[9E+09,9E+09,9E+09,9E+09,9E+09,9E+09]];
CONST robtarget LHP_415:=[[1568.58,736.45,-284.14],[0.571745,-0.00397095,-0.00657964,-0.820396],[-1,0,-1,0],[9E+09,9E+09,9E+09,9E+09,9E+09,9E+09]];
CONST robtarget LHP_420:=[[1508.30,917.00,-395.22],[0.556499,0.0508994,0.0317793,-0.828678],[-1,-1,-1,0],[9E+09,9E+09,9E+09,9E+09,9E+09,9E+09]];
CONST robtarget LHP_425:=[[1495.25,987.39,-357.83],[0.551104,0.0895725,0.0518729,-0.827992],[-1,-1,-1,0],[9E+09,9E+09,9E+09,9E+09,9E+09,9E+09]];
CONST robtarget LHP_430:=[[1328.35,635.44,-278.20],[0.501405,0.0212305,0.11734,-0.856956],[-1,-1,0,0],[9E+09,9E+09,9E+09,9E+09,9E+09,9E+09]];
CONST robtarget LHP_435:=[[1126.70,526.89,-238.13],[0.384755,0.0646485,0.107006,-0.914513],[-1,-1,0,0],[9E+09,9E+09,9E+09,9E+09,9E+09,9E+09]];
CONST robtarget LHP_440:=[[1126.70,526.87,-238.14],[0.384757,0.0646487,0.107006,-0.914512],[-1,-1,0,0],[9E+09,9E+09,9E+09,9E+09,9E+09,9E+09]];
CONST robtarget LHP_445:=[[1328.35,635.43,-278.21],[0.501406,0.0212292,0.11734,-0.856956],[-1,-1,0,0],[9E+09,9E+09,9E+09,9E+09,9E+09,9E+09]];
CONST robtarget LHP_450:=[[1495.26,987.39,-357.84],[0.551103,0.0895724,0.0518701,-0.827993],[-1,-1,-1,0],[9E+09,9E+09,9E+09,9E+09,9E+09,9E+09]];
CONST robtarget LHP_455:=[[1606.25,805.30,-336.47],[0.591189,0.0705667,0.0504833,-0.801852],[-1,-1,-1,0],[9E+09,9E+09,9E+09,9E+09,9E+09,9E+09]];
CONST robtarget LHP_460:=[[1846.21,646.41,-266.45],[0.66313,0.055392,0.0578373,-0.744207],[-1,-1,-1,0],[9E+09,9E+09,9E+09,9E+09,9E+09,9E+09]];
CONST robtarget LHP_465:=[[1831.93,634.62,-78.38],[0.625946,0.00957367,0.0100376,-0.779743],[-1,-1,-1,0],[9E+09,9E+09,9E+09,9E+09,9E+09,9E+09]];
CONST robtarget LHP_470:=[[1778.25,512.89,-42.92],[0.553639,0.000122695,-2.9028E-05,-0.832757],[-1,-1,-1,0],[9E+09,9E+09,9E+09,9E+09,9E+09,9E+09]];
CONST robtarget LHP_475:=[[1581.22,548.75,-125.86],[0.508525,0.0149425,0.00198371,-0.860915],[-1,0,-1,0],[9E+09,9E+09,9E+09,9E+09,9E+09,9E+09]];
CONST robtarget LHP_480:=[[1526.71,530.36,-111.44],[0.495097,0.0157343,0.00230728,-0.868692],[-1,0,-1,0],[9E+09,9E+09,9E+09,9E+09,9E+09,9E+09]];
CONST robtarget LHP_485:=[[1496.52905,533.620972,-169.427002],[0.5015252,0.014323151,0.035049833,-0.8643141],[-1,-1,-1,0],[9E9,9E9,9E9,9E9,9E9,9E9]];
CONST robtarget LHP_490:=[[1628.88,359.00,-167.42],[0.509965,0.00587853,-0.00326077,-0.860169],[-1,0,-1,0],[9E+09,9E+09,9E+09,9E+09,9E+09,9E+09]];
CONST robtarget LHP_495:=[[1653.10,363.04,-167.43],[0.50985,0.0307676,0.0114918,-0.859636],[-1,0,-1,0],[9E+09,9E+09,9E+09,9E+09,9E+09,9E+09]];
CONST robtarget LHP_500:=[[1734.14,581.56,-229.81],[0.51369,0.0926739,0.046858,-0.851668],[-1,-1,-1,0],[9E+09,9E+09,9E+09,9E+09,9E+09,9E+09]];
CONST robtarget LHP_505:=[[1850.77,754.32,-287.10],[0.562259,0.138379,0.0973397,-0.809469],[-1,-1,-1,0],[9E+09,9E+09,9E+09,9E+09,9E+09,9E+09]];
CONST robtarget LHP_510:=[[1850.71,883.30,-361.37],[0.589549,0.148661,0.155296,-0.778598],[-1,-1,-1,0],[9E+09,9E+09,9E+09,9E+09,9E+09,9E+09]];
CONST robtarget LHP_515:=[[1850.60,911.16,-304.76],[0.610795,0.143869,0.202267,-0.751877],[-1,-1,-1,0],[9E+09,9E+09,9E+09,9E+09,9E+09,9E+09]];
CONST robtarget LHP_520:=[[1845.93,938.54,-187.19],[0.617535,0.126482,0.223985,-0.743292],[-1,-1,-1,0],[9E+09,9E+09,9E+09,9E+09,9E+09,9E+09]];
CONST robtarget LHP_525:=[[1839.91,764.25,251.37],[0.609113,0.0794277,0.135403,-0.777392],[-1,-1,-1,0],[9E+09,9E+09,9E+09,9E+09,9E+09,9E+09]];
CONST robtarget LHP_530:=[[1951.53,815.35,1215.32],[0.610126,-0.0704393,-0.00824645,-0.789124],[-1,0,-1,0],[9E+09,9E+09,9E+09,9E+09,9E+09,9E+09]];
CONST robtarget LHP_535:=[[2438.93,960.39,2235.39],[0.671457,-0.189483,-0.125804,-0.705277],[-1,0,-1,0],[9E+09,9E+09,9E+09,9E+09,9E+09,9E+09]];

! ------------------------------------------------------------
  ! Unterprogramm:
  ! Stand
  ! Daimler AG - Werk Ludwigsfelde
  ! ------------------------------------------------------------
  ! ************************************************************
  ! Kommentar: Achtung
  !            automatisch generiert!!!!!!!!!!!!!!!!!!
  ! ************************************************************

! Robotername:            1606R04
! Anlagenbezeichn:        Linie 16          Stations-Nr:  1606
! Stand / Version:        04.08.2009 / 1.1
! Name Bearbeiter:        Karmann
! Applikationssteuerung:  Punktschweissen
! Baumuster:              FHL T1 R2


INIT_SW_BASE;

WKZ_1_AUFNEHMEN;

MoveJ ToolHome1,vSchnell,fine,nomtcp1;

MoveJ LHP_000,vSchnell,fine,nomtcp1\WObj:=BS_1606_1A;

Vorhub\auf;

ABL 2\ABL_WAIT;
ABL 10\ABL_SET;

!1606R04_1606R06
KOLLISION_ZONE 2\Anfrage;
!1606R04_1606R06
KOLLISION_ZONE 7\Anfrage;
!1606R04_1606R06
KOLLISION_ZONE 9\Anfrage;


!!
! ZMIANA Kolejnosci
! Zrobic dojazd
!
WaitUntil FALSE;

MoveJ LHP_125,vSchnell,z100,nomtcp1\WObj:=BS_1606_1A;
!

SpotL G0216190478BP20\VFO:=210\Vorhub_Auf,vSpot,nomtcp1\WObj:=BS_1606_1A;
SpotL G0216190582BP20\VFO:=210\Vorhub_Auf,vSpot,nomtcp1\WObj:=BS_1606_1A;

! Zrobic dojazd
WaitUntil FALSE;
MoveJ LHP_130,vSchnell,z100,nomtcp1\WObj:=BS_1606_1A;
MoveJ LHP_135,vSchnell,z1,nomtcp1\WObj:=BS_1606_1A;
MoveL LHP_140,vSchnell,z1,nomtcp1\WObj:=BS_1606_1A;
MoveL LHP_145,vSchnell,z1,nomtcp1\WObj:=BS_1606_1A;
SpotL G0216190492BP20\VFO:=210\Vorhub_Auf,vSpot,nomtcp1\WObj:=BS_1606_1A;

WaitUntil FALSE;
!
! Zrobic dojazd
!

!1606R04_1606R06
KOLLISION_ZONE 2\Freigabe;

MoveJ LHP_480, vSchnell, z100, nomtcp1\WObj:=BS_1606_1A;

SpotL G0216190576BP20\VFO:=210,vSpot,nomtcp1\WObj:=BS_1606_1A;
SpotL G0213198812BP20\VFO:=210\Vorhub_Auf,vSpot,nomtcp1\WObj:=BS_1606_1A;

!
! Zrobic dojazd
!
WaitUntil FALSE;

SpotL G0213198810BP20\VFO:=210,vSpot,nomtcp1\WObj:=BS_1606_1A;
SpotL G0213198808BP20\VFO:=210,vSpot,nomtcp1\WObj:=BS_1606_1A;
SpotL G0216021970BP20\VFO:=210,vSpot,nomtcp1\WObj:=BS_1606_1A;

!
! zrobic dojazd
!
WaitUntil false;

MoveJ LHP_470,vSchnell,fine,nomtcp1\WObj:=BS_1606_1A;

SpotL G0216021972BP20\VFO:=210,vSpot,nomtcp1\WObj:=BS_1606_1A;

MoveJ LHP_485,vSchnell,z100,nomtcp1\WObj:=BS_1606_1A;

SpotL G0216021974BP20\VFO:=210,vSpot,nomtcp1\WObj:=BS_1606_1A;

MoveJ LHP_190,vSchnell,z100,nomtcp1\WObj:=BS_1606_1A;
MoveJ LHP_195,vSchnell,z100,nomtcp1\WObj:=BS_1606_1A;

SpotL G0216022098BP20\VFO:=210\Vorhub_Auf,vSpot,nomtcp1\WObj:=BS_1606_1A;

!
! zrobic dojazd
!
WaitUntil FALSE;

MoveJ LHP_035,vSchnell,z100,nomtcp1\WObj:=BS_1606_1A;

SpotL G0216022096BP20\VFO:=210,vSpot,nomtcp1\WObj:=BS_1606_1A;
SpotL G0216022094BP20\VFO:=210,vSpot,nomtcp1\WObj:=BS_1606_1A;

!
! zrobic dojazd
!
waituntil FALSE;

MoveJ LHP_465,vSchnell,z100,nomtcp1\WObj:=BS_1606_1A;

SpotL G0216021976BP20\VFO:=210,vSpot,nomtcp1\WObj:=BS_1606_1A;
SpotL G0216190440BP20\VFO:=210,vSpot,nomtcp1\WObj:=BS_1606_1A;
SpotL G0216190438BP20\VFO:=210,vSpot,nomtcp1\WObj:=BS_1606_1A;
SpotL G0216190436BP20\VFO:=210,vSpot,nomtcp1\WObj:=BS_1606_1A;

!
! zrobic dojazd
!
WaitUntil FALSE;

MoveJ LHP_475,vSchnell,z100,nomtcp1\WObj:=BS_1606_1A;

SpotL G0216190434BP20\VFO:=210\Vorhub_Auf,vSpot,nomtcp1\WObj:=BS_1606_1A;
SpotL G0216190432BP20\VFO:=210,vSpot,nomtcp1\WObj:=BS_1606_1A;
SpotL G0216190430BP20\VFO:=210,vSpot,nomtcp1\WObj:=BS_1606_1A;
SpotL G0216190428BP20\VFO:=210,vSpot,nomtcp1\WObj:=BS_1606_1A;

MoveJ LHP_460,vSchnell,z100,nomtcp1\WObj:=BS_1606_1A;

!
! zrobic dojazd
!
WaitUntil FALSE;

MoveJ LHP_230,vSchnell,z100,nomtcp1\WObj:=BS_1606_1A;

SpotL G0216190446BP20\VFO:=210\Vorhub_Auf,vSpot,nomtcp1\WObj:=BS_1606_1A;

KOLLISION_ZONE 1\Anfrage;
KOLLISION_ZONE 6\Anfrage;

!
! zrobic dojazd
!
WaitUntil FALSE;


MoveJ LHP_235,vSchnell,z100,nomtcp1\WObj:=BS_1606_1A;
MoveJ LHP_240,vSchnell,z100,nomtcp1\WObj:=BS_1606_1A;
MoveJ LHP_245,vSchnell,z100,nomtcp1\WObj:=BS_1606_1A;
MoveJ LHP_250,vSchnell,z100,nomtcp1\WObj:=BS_1606_1A;
MoveJ LHP_255,vSchnell,z100,nomtcp1\WObj:=BS_1606_1A;
MoveJ LHP_260,vSchnell,z100,nomtcp1\WObj:=BS_1606_1A;
MoveJ LHP_265,vSchnell,z100,nomtcp1\WObj:=BS_1606_1A;
MoveJ LHP_270,vSchnell,z100,nomtcp1\WObj:=BS_1606_1A;
MoveJ LHP_275,vSchnell,z100,nomtcp1\WObj:=BS_1606_1A;
MoveJ LHP_280,vSchnell,z100,nomtcp1\WObj:=BS_1606_1A;
MoveL LHP_285,vSchnell,z5,nomtcp1\WObj:=BS_1606_1A;
MoveL LHP_290,vSchnell,z5,nomtcp1\WObj:=BS_1606_1A;
MoveL LHP_295,vSchnell,z5,nomtcp1\WObj:=BS_1606_1A;
MoveL LHP_300,vSchnell,z5,nomtcp1\WObj:=BS_1606_1A;
MoveL LHP_305,vSchnell,z5,nomtcp1\WObj:=BS_1606_1A;

SpotL G0216190480BP20\VFO:=210\Vorhub_Auf, vSpot, nomtcp1\WObj:=BS_1606_1A;

MoveL LHP_310,vSchnell,z5,nomtcp1\WObj:=BS_1606_1A;
MoveL LHP_315,vSchnell,z5,nomtcp1\WObj:=BS_1606_1A;
MoveL LHP_320,vSchnell,z5,nomtcp1\WObj:=BS_1606_1A;
MoveL LHP_325,vSchnell,z5,nomtcp1\WObj:=BS_1606_1A;
MoveL LHP_330,vSchnell,z5,nomtcp1\WObj:=BS_1606_1A;
MoveL LHP_335,vSchnell,z5,nomtcp1\WObj:=BS_1606_1A;
MoveL LHP_340,vSchnell,z5,nomtcp1\WObj:=BS_1606_1A;

SpotL G0216022394BP20\VFO:=210\Vorhub_Auf,vSpot,nomtcp1\WObj:=BS_1606_1A;

MoveJ LHP_345,vSchnell,z100,nomtcp1\WObj:=BS_1606_1A;
MoveJ LHP_350,vSchnell,fine,nomtcp1\WObj:=BS_1606_1A;


SpotL G0216022386BP20\VFO:=210,vSpot,nomtcp1\WObj:=BS_1606_1A;
SpotL G0216047033BP20\VFO:=210,vSpot,nomtcp1\WObj:=BS_1606_1A;

KOLLISION_ZONE 6\Freigabe;

SpotL G0216047032BP20\VFO:=210\Vorhub_Auf,vSpot,nomtcp1\WObj:=BS_1606_1A;

MoveJ LHP_355,vSchnell,z100,nomtcp1\WObj:=BS_1606_1A;
MoveJ LHP_360,vSchnell,z100,nomtcp1\WObj:=BS_1606_1A;
MoveJ LHP_365,vSchnell,z100,nomtcp1\WObj:=BS_1606_1A;
MoveJ LHP_370,vSchnell,z100,nomtcp1\WObj:=BS_1606_1A;

!
! zrobic dojazd
!
WaitUntil FALSE;

MoveJ LHP_430,vSchnell,z100,nomtcp1\WObj:=BS_1606_1A;
MoveJ LHP_435,vSchnell,z100,nomtcp1\WObj:=BS_1606_1A;

SpotL G0216047028BP20\VFO:=210,vSpot,nomtcp1\WObj:=BS_1606_1A;
SpotL G0216047029BP20\VFO:=210,vSpot,nomtcp1\WObj:=BS_1606_1A;
SpotL G0216022368BP20\VFO:=210,vSpot,nomtcp1\WObj:=BS_1606_1A;
SpotL G0216022370BP20\VFO:=210\Vorhub_Auf,vSpot,nomtcp1\WObj:=BS_1606_1A;

MoveJ LHP_440,vSchnell,z100,nomtcp1\WObj:=BS_1606_1A;
MoveJ LHP_445,vSchnell,z100,nomtcp1\WObj:=BS_1606_1A;
MoveJ LHP_450,vSchnell,z100,nomtcp1\WObj:=BS_1606_1A;
MoveJ LHP_455,vSchnell,z100,nomtcp1\WObj:=BS_1606_1A;

!
! zrobic dojazd
!
WaitUntil FALSE;

MoveJ LHP_040,vSchnell,z100,nomtcp1\WObj:=BS_1606_1A;

SpotL G0216190516BP20\VFO:=210,vSpot,nomtcp1\WObj:=BS_1606_1A;

KOLLISION_ZONE 1\Freigabe;
KOLLISION_ZONE 7\Freigabe;
KOLLISION_ZONE 8\Anfrage;

MoveJ LHP_045,vSchnell,z100,nomtcp1\WObj:=BS_1606_1A;

SpotL G0216190518BP20\VFO:=210,vSpot,nomtcp1\WObj:=BS_1606_1A;
SpotL G0216190520BP20\VFO:=210,vSpot,nomtcp1\WObj:=BS_1606_1A;

MoveJ LHP_050,vSchnell,z100,nomtcp1\WObj:=BS_1606_1A;

SpotL G0216190522BP20\VFO:=210,vSpot,nomtcp1\WObj:=BS_1606_1A;
SpotL G0216190524BP20\VFO:=210,vSpot,nomtcp1\WObj:=BS_1606_1A;

!1606R04_1606R03
KOLLISION_ZONE 4\Anfrage;

SpotL G0216190526BP20\VFO:=210,vSpot,nomtcp1\WObj:=BS_1606_1A;
SpotL G0216190528BP20\VFO:=210\Vorhub_Auf,vSpot,nomtcp1\WObj:=BS_1606_1A;

MoveJ LHP_055,vSchnell,z100,nomtcp1\WObj:=BS_1606_1A;
MoveJ LHP_060,vSchnell,z100,nomtcp1\WObj:=BS_1606_1A;
MoveJ LHP_065,vSchnell,z100,nomtcp1\WObj:=BS_1606_1A;
MoveJ LHP_070,vSchnell,z100,nomtcp1\WObj:=BS_1606_1A;
MoveJ LHP_075,vSchnell,z100,nomtcp1\WObj:=BS_1606_1A;
MoveJ LHP_080,vSchnell,z100,nomtcp1\WObj:=BS_1606_1A;

SpotL G0216190508BP20\VFO:=210,vSpot,nomtcp1\WObj:=BS_1606_1A;

MoveJ LHP_085,vSchnell,z100,nomtcp1\WObj:=BS_1606_1A;

!
! zrobic dojazd
!
WaitUntil FALSE;

MoveJ LHP_400,vSchnell,z100,nomtcp1\WObj:=BS_1606_1A;

SpotL G0216190500BP20\VFO:=210\Vorhub_Auf,vSpot,nomtcp1\WObj:=BS_1606_1A;

MoveJ LHP_405,vSchnell,z100,nomtcp1\WObj:=BS_1606_1A;

!
! zrobic dojazd
!
WaitUntil FALSE;

MoveJ LHP_020,vSchnell,z100,nomtcp1\WObj:=BS_1606_1A;
MoveJ LHP_025,vSchnell,z100,nomtcp1\WObj:=BS_1606_1A;
MoveJ LHP_030,vSchnell,z100,nomtcp1\WObj:=BS_1606_1A;
MoveJ LHP_090,vSchnell,z100,nomtcp1\WObj:=BS_1606_1A;

SpotL G0216190506BP20\VFO:=210\Vorhub_Auf,vSpot,nomtcp1\WObj:=BS_1606_1A;

!
! zrobic dojazd
!
WaitUntil FALSE;

MoveJ LHP_390,vSchnell,fine,nomtcp1\WObj:=BS_1606_1A;


SpotL G0216190498BP20\VFO:=210,vSpot,nomtcp1\WObj:=BS_1606_1A;

MoveJ LHP_395,vSchnell,z100,nomtcp1\WObj:=BS_1606_1A;

SpotL G0216190488BP20\VFO:=210,vSpot,nomtcp1\WObj:=BS_1606_1A;

MoveJ LHP_410,vSchnell,z100,nomtcp1\WObj:=BS_1606_1A;

SpotL G0216190496BP20\VFO:=210,vSpot,nomtcp1\WObj:=BS_1606_1A;
SpotL G0216190494BP20\VFO:=210,vSpot,nomtcp1\WObj:=BS_1606_1A;

!
! zrobic dojazd
!
WaitUntil FALSE;

MoveJ LHP_215,vSchnell,z100,nomtcp1\WObj:=BS_1606_1A;

SpotL G0216190502BP20\VFO:=210\Vorhub_Auf,vSpot,nomtcp1\WObj:=BS_1606_1A;

KOLLISION_ZONE 8\Freigabe;

!
! zrobic dojazd
!
WaitUntil FALSE;

MoveJ LHP_220,vSchnell,z100,nomtcp1\WObj:=BS_1606_1A;

SpotL G0213198814BP20\VFO:=210\Vorhub_Auf,vSpot,nomtcp1\WObj:=BS_1606_1A;

MoveJ LHP_225,vSchnell,z100,nomtcp1\WObj:=BS_1606_1A;

!
! zrobic dojazd
!
WaitUntil FALSE;

MoveJ LHP_490,vSchnell,z100,nomtcp1\WObj:=BS_1606_1A;

SpotL G0213198816BP20\VFO:=210,vSpot,nomtcp1\WObj:=BS_1606_1A;
SpotL G0213198818BP20\VFO:=210\Vorhub_Auf,vSpot,nomtcp1\WObj:=BS_1606_1A;

MoveJ LHP_495, vSchnell,z100,nomtcp1\WObj:=BS_1606_1A;
MoveJ LHP_500, vSchnell,z10,nomtcp1\WObj:=BS_1606_1A;

!
! zrobic dojazd
!
WaitUntil FALSE;

MoveJ LHP_205,vSchnell,z100,nomtcp1\WObj:=BS_1606_1A;
MoveJ LHP_210,vSchnell,fine,nomtcp1\WObj:=BS_1606_1A;


SpotL G0216022102BP20\VFO:=210,vSpot,nomtcp1\WObj:=BS_1606_1A;
SpotL G0216022100BP20\VFO:=210,vSpot,nomtcp1\WObj:=BS_1606_1A;

MoveJ LHP_375,vSchnell,z100,nomtcp1\WObj:=BS_1606_1A;
MoveJ LHP_380,vSchnell,z100,nomtcp1\WObj:=BS_1606_1A;

!
! powrot do home
!
WaitUntil FALSE;


!1606R04_1606R03
KOLLISION_ZONE 4\Freigabe;

MoveJ LHP_535,vSchnell,z100,nomtcp1\WObj:=BS_1606_1A;

MoveJ ToolHome1,vSchnell,fine,nomtcp1;

!1606R04_1606R06
KOLLISION_ZONE 1\Freigabe;
KOLLISION_ZONE 9\Freigabe;


ABL 254\ABL_WAIT;
ABL 255\ABL_SET;

!
ENDPROC

PROC swp_223300_0_st1606_1()

